   1:  PR[GP1:91,1] = PR[GP1:90,1] + 33.449;
   1:  PR[GP1:91,2] = PR[GP1:90,2] + -36.632;
   1:L PR[91] 10mm/sec CNT100;
   1:  PR[GP1:91,1] = PR[GP1:90,1] + 41.672;
   1:  PR[GP1:91,2] = PR[GP1:90,2] + -33.015;
   1:L PR[91] 10mm/sec CNT100;
   1:  PR[GP1:91,1] = PR[GP1:90,1] + 44.293;
   1:  PR[GP1:91,2] = PR[GP1:90,2] + -31.371;
   1:L PR[91] 10mm/sec CNT100;
   1:  PR[GP1:91,1] = PR[GP1:90,1] + 46.699;
   1:  PR[GP1:91,2] = PR[GP1:90,2] + -29.026;
   1:L PR[91] 10mm/sec CNT100;
   1:  PR[GP1:91,1] = PR[GP1:90,1] + 52.748;
   1:  PR[GP1:91,2] = PR[GP1:90,2] + -23.523;
   1:L PR[91] 10mm/sec CNT100;
   1:  PR[GP1:91,1] = PR[GP1:90,1] + 54.691;
   1:  PR[GP1:91,2] = PR[GP1:90,2] + -20.511;
   1:L PR[91] 10mm/sec CNT100;
   1:  PR[GP1:91,1] = PR[GP1:90,1] + 58.358;
   1:  PR[GP1:91,2] = PR[GP1:90,2] + -13.882;
   1:L PR[91] 10mm/sec CNT100;
   1:  PR[GP1:91,1] = PR[GP1:90,1] + 59.590;
   1:  PR[GP1:91,2] = PR[GP1:90,2] + -10.532;
   1:L PR[91] 10mm/sec CNT100;
   1:  PR[GP1:91,1] = PR[GP1:90,1] + 60.008;
   1:  PR[GP1:91,2] = PR[GP1:90,2] + -6.857;
   1:L PR[91] 10mm/sec CNT100;
   1:  PR[GP1:91,1] = PR[GP1:90,1] + 61.228;
   1:  PR[GP1:91,2] = PR[GP1:90,2] + 0.296;
   1:L PR[91] 10mm/sec CNT100;
   1:  PR[GP1:91,1] = PR[GP1:90,1] + 60.818;
   1:  PR[GP1:91,2] = PR[GP1:90,2] + 3.922;
   1:L PR[91] 10mm/sec CNT100;
   1:  PR[GP1:91,1] = PR[GP1:90,1] + 59.591;
   1:  PR[GP1:91,2] = PR[GP1:90,2] + 11.088;
   1:L PR[91] 10mm/sec CNT100;
   1:  PR[GP1:91,1] = PR[GP1:90,1] + 58.352;
   1:  PR[GP1:91,2] = PR[GP1:90,2] + 14.455;
   1:L PR[91] 10mm/sec CNT100;
   1:  PR[GP1:91,1] = PR[GP1:90,1] + 54.670;
   1:  PR[GP1:91,2] = PR[GP1:90,2] + 21.095;
   1:L PR[91] 10mm/sec CNT100;
   1:  PR[GP1:91,1] = PR[GP1:90,1] + 52.721;
   1:  PR[GP1:91,2] = PR[GP1:90,2] + 24.118;
   1:L PR[91] 10mm/sec CNT100;
   1:  PR[GP1:91,1] = PR[GP1:90,1] + 50.377;
   1:  PR[GP1:91,2] = PR[GP1:90,2] + 26.413;
   1:L PR[91] 10mm/sec CNT100;
   1:  PR[GP1:91,1] = PR[GP1:90,1] + 44.256;
   1:  PR[GP1:91,2] = PR[GP1:90,2] + 31.953;
   1:L PR[91] 10mm/sec CNT100;
   1:  PR[GP1:91,1] = PR[GP1:90,1] + 41.625;
   1:  PR[GP1:91,2] = PR[GP1:90,2] + 33.604;
   1:L PR[91] 10mm/sec CNT100;
   1:  PR[GP1:91,1] = PR[GP1:90,1] + 33.371;
   1:  PR[GP1:91,2] = PR[GP1:90,2] + 37.210;
   1:L PR[91] 10mm/sec CNT100;
   1:  PR[GP1:91,1] = PR[GP1:90,1] + 30.668;
   1:  PR[GP1:91,2] = PR[GP1:90,2] + 38.196;
   1:L PR[91] 10mm/sec CNT100;
   1:  PR[GP1:91,1] = PR[GP1:90,1] + 28.112;
   1:  PR[GP1:91,2] = PR[GP1:90,2] + 38.559;
   1:L PR[91] 10mm/sec CNT100;
   1:  PR[GP1:91,1] = PR[GP1:90,1] + 18.357;
   1:  PR[GP1:91,2] = PR[GP1:90,2] + 39.465;
   1:L PR[91] 10mm/sec CNT100;
   1:  PR[GP1:91,1] = PR[GP1:90,1] + 16.104;
   1:  PR[GP1:91,2] = PR[GP1:90,2] + 39.316;
   1:L PR[91] 10mm/sec CNT100;
   1:  PR[GP1:91,1] = PR[GP1:90,1] + 5.716;
   1:  PR[GP1:91,2] = PR[GP1:90,2] + 36.862;
   1:L PR[91] 10mm/sec CNT100;
   1:  PR[GP1:91,1] = PR[GP1:90,1] + 3.913;
   1:  PR[GP1:91,2] = PR[GP1:90,2] + 36.344;
   1:L PR[91] 10mm/sec CNT100;
   1:  PR[GP1:91,1] = PR[GP1:90,1] + 1.574;
   1:  PR[GP1:91,2] = PR[GP1:90,2] + 35.102;
   1:L PR[91] 10mm/sec CNT100;
   1:  PR[GP1:91,1] = PR[GP1:90,1] + -0.263;
   1:  PR[GP1:91,2] = PR[GP1:90,2] + 33.609;
   1:L PR[91] 10mm/sec CNT100;
   1:  PR[GP1:91,1] = PR[GP1:90,1] + -2.096;
   1:  PR[GP1:91,2] = PR[GP1:90,2] + 35.099;
   1:L PR[91] 10mm/sec CNT100;
   1:  PR[GP1:91,1] = PR[GP1:90,1] + -4.438;
   1:  PR[GP1:91,2] = PR[GP1:90,2] + 36.345;
   1:L PR[91] 10mm/sec CNT100;
   1:  PR[GP1:91,1] = PR[GP1:90,1] + -6.237;
   1:  PR[GP1:91,2] = PR[GP1:90,2] + 36.862;
   1:L PR[91] 10mm/sec CNT100;
   1:  PR[GP1:91,1] = PR[GP1:90,1] + -16.629;
   1:  PR[GP1:91,2] = PR[GP1:90,2] + 39.315;
   1:L PR[91] 10mm/sec CNT100;
   1:  PR[GP1:91,1] = PR[GP1:90,1] + -18.875;
   1:  PR[GP1:91,2] = PR[GP1:90,2] + 39.464;
   1:L PR[91] 10mm/sec CNT100;
   1:  PR[GP1:91,1] = PR[GP1:90,1] + -21.435;
   1:  PR[GP1:91,2] = PR[GP1:90,2] + 39.109;
   1:L PR[91] 10mm/sec CNT100;
   1:  PR[GP1:91,1] = PR[GP1:90,1] + -31.222;
   1:  PR[GP1:91,2] = PR[GP1:90,2] + 38.189;
   1:L PR[91] 10mm/sec CNT100;
   1:  PR[GP1:91,1] = PR[GP1:90,1] + -33.908;
   1:  PR[GP1:91,2] = PR[GP1:90,2] + 37.206;
   1:L PR[91] 10mm/sec CNT100;
   1:  PR[GP1:91,1] = PR[GP1:90,1] + -42.162;
   1:  PR[GP1:91,2] = PR[GP1:90,2] + 33.597;
   1:L PR[91] 10mm/sec CNT100;
   1:  PR[GP1:91,1] = PR[GP1:90,1] + -44.799;
   1:  PR[GP1:91,2] = PR[GP1:90,2] + 31.934;
   1:L PR[91] 10mm/sec CNT100;
   1:  PR[GP1:91,1] = PR[GP1:90,1] + -47.210;
   1:  PR[GP1:91,2] = PR[GP1:90,2] + 29.580;
   1:L PR[91] 10mm/sec CNT100;
   1:  PR[GP1:91,1] = PR[GP1:90,1] + -53.284;
   1:  PR[GP1:91,2] = PR[GP1:90,2] + 24.081;
   1:L PR[91] 10mm/sec CNT100;
   1:  PR[GP1:91,1] = PR[GP1:90,1] + -55.205;
   1:  PR[GP1:91,2] = PR[GP1:90,2] + 21.082;
   1:L PR[91] 10mm/sec CNT100;
   1:  PR[GP1:91,1] = PR[GP1:90,1] + -58.888;
   1:  PR[GP1:91,2] = PR[GP1:90,2] + 14.430;
   1:L PR[91] 10mm/sec CNT100;
   1:  PR[GP1:91,1] = PR[GP1:90,1] + -60.126;
   1:  PR[GP1:91,2] = PR[GP1:90,2] + 11.020;
   1:L PR[91] 10mm/sec CNT100;
   1:  PR[GP1:91,1] = PR[GP1:90,1] + -60.529;
   1:  PR[GP1:91,2] = PR[GP1:90,2] + 7.423;
   1:L PR[91] 10mm/sec CNT100;
   1:  PR[GP1:91,1] = PR[GP1:90,1] + -61.754;
   1:  PR[GP1:91,2] = PR[GP1:90,2] + 0.261;
   1:L PR[91] 10mm/sec CNT100;
   1:  PR[GP1:91,1] = PR[GP1:90,1] + -61.359;
   1:  PR[GP1:91,2] = PR[GP1:90,2] + -3.287;
   1:L PR[91] 10mm/sec CNT100;
   1:  PR[GP1:91,1] = PR[GP1:90,1] + -60.137;
   1:  PR[GP1:91,2] = PR[GP1:90,2] + -10.430;
   1:L PR[91] 10mm/sec CNT100;
   1:  PR[GP1:91,1] = PR[GP1:90,1] + -58.893;
   1:  PR[GP1:91,2] = PR[GP1:90,2] + -13.857;
   1:L PR[91] 10mm/sec CNT100;
   1:  PR[GP1:91,1] = PR[GP1:90,1] + -55.226;
   1:  PR[GP1:91,2] = PR[GP1:90,2] + -20.497;
   1:L PR[91] 10mm/sec CNT100;
   1:  PR[GP1:91,1] = PR[GP1:90,1] + -53.299;
   1:  PR[GP1:91,2] = PR[GP1:90,2] + -23.506;
   1:L PR[91] 10mm/sec CNT100;
   1:  PR[GP1:91,1] = PR[GP1:90,1] + -50.951;
   1:  PR[GP1:91,2] = PR[GP1:90,2] + -25.809;
   1:L PR[91] 10mm/sec CNT100;
   1:  PR[GP1:91,1] = PR[GP1:90,1] + -44.856;
   1:  PR[GP1:91,2] = PR[GP1:90,2] + -31.339;
   1:L PR[91] 10mm/sec CNT100;
   1:  PR[GP1:91,1] = PR[GP1:90,1] + -42.208;
   1:  PR[GP1:91,2] = PR[GP1:90,2] + -33.008;
   1:L PR[91] 10mm/sec CNT100;
   1:  PR[GP1:91,1] = PR[GP1:90,1] + -33.986;
   1:  PR[GP1:91,2] = PR[GP1:90,2] + -36.627;
   1:L PR[91] 10mm/sec CNT100;
   1:  PR[GP1:91,1] = PR[GP1:90,1] + -31.287;
   1:  PR[GP1:91,2] = PR[GP1:90,2] + -37.616;
   1:L PR[91] 10mm/sec CNT100;
   1:  PR[GP1:91,1] = PR[GP1:90,1] + -28.722;
   1:  PR[GP1:91,2] = PR[GP1:90,2] + -37.981;
   1:L PR[91] 10mm/sec CNT100;
   1:  PR[GP1:91,1] = PR[GP1:90,1] + -18.999;
   1:  PR[GP1:91,2] = PR[GP1:90,2] + -38.913;
   1:L PR[91] 10mm/sec CNT100;
   1:  PR[GP1:91,1] = PR[GP1:90,1] + -16.737;
   1:  PR[GP1:91,2] = PR[GP1:90,2] + -38.764;
   1:L PR[91] 10mm/sec CNT100;
   1:  PR[GP1:91,1] = PR[GP1:90,1] + -6.516;
   1:  PR[GP1:91,2] = PR[GP1:90,2] + -36.426;
   1:L PR[91] 10mm/sec CNT100;
   1:  PR[GP1:91,1] = PR[GP1:90,1] + -4.644;
   1:  PR[GP1:91,2] = PR[GP1:90,2] + -35.888;
   1:L PR[91] 10mm/sec CNT100;
   1:  PR[GP1:91,1] = PR[GP1:90,1] + -0.265;
   1:  PR[GP1:91,2] = PR[GP1:90,2] + -33.323;
   1:L PR[91] 10mm/sec CNT100;
   1:  PR[GP1:91,1] = PR[GP1:90,1] + 3.860;
   1:  PR[GP1:91,2] = PR[GP1:90,2] + -35.957;
   1:  PR[GP1:91,3] = PR[GP1:90,3] + 75.335;
   1:L PR[91] 10mm/sec CNT100;
   1:  PR[GP1:91,1] = PR[GP1:90,1] + 5.615;
   1:  PR[GP1:91,2] = PR[GP1:90,2] + -36.460;
   1:L PR[91] 10mm/sec CNT100;
   1:  PR[GP1:91,1] = PR[GP1:90,1] + 16.035;
   1:  PR[GP1:91,2] = PR[GP1:90,2] + -38.845;
   1:L PR[91] 10mm/sec CNT100;
   1:  PR[GP1:91,1] = PR[GP1:90,1] + 18.154;
   1:  PR[GP1:91,2] = PR[GP1:90,2] + -38.985;
   1:L PR[91] 10mm/sec CNT100;
   1:  PR[GP1:91,1] = PR[GP1:90,1] + 20.568;
   1:  PR[GP1:91,2] = PR[GP1:90,2] + -38.652;
   1:L PR[91] 10mm/sec CNT100;
   1:  PR[GP1:91,1] = PR[GP1:90,1] + 30.542;
   1:  PR[GP1:91,2] = PR[GP1:90,2] + -37.683;
   1:L PR[91] 10mm/sec CNT100;
   1:  PR[GP1:91,1] = PR[GP1:90,1] + 33.105;
   1:  PR[GP1:91,2] = PR[GP1:90,2] + -36.747;
   1:L PR[91] 10mm/sec CNT100;
   1:  PR[GP1:91,1] = PR[GP1:90,1] + 41.526;
   1:  PR[GP1:91,2] = PR[GP1:90,2] + -33.044;
   1:L PR[91] 10mm/sec CNT100;
   1:  PR[GP1:91,1] = PR[GP1:90,1] + 44.038;
   1:  PR[GP1:91,2] = PR[GP1:90,2] + -31.468;
   1:L PR[91] 10mm/sec CNT100;
   1:  PR[GP1:91,1] = PR[GP1:90,1] + 46.343;
   1:  PR[GP1:91,2] = PR[GP1:90,2] + -29.221;
   1:L PR[91] 10mm/sec CNT100;
   1:  PR[GP1:91,1] = PR[GP1:90,1] + 52.561;
   1:  PR[GP1:91,2] = PR[GP1:90,2] + -23.565;
   1:L PR[91] 10mm/sec CNT100;
   1:  PR[GP1:91,1] = PR[GP1:90,1] + 54.429;
   1:  PR[GP1:91,2] = PR[GP1:90,2] + -20.668;
   1:L PR[91] 10mm/sec CNT100;
   1:  PR[GP1:91,1] = PR[GP1:90,1] + 58.203;
   1:  PR[GP1:91,2] = PR[GP1:90,2] + -13.846;
   1:L PR[91] 10mm/sec CNT100;
   1:  PR[GP1:91,1] = PR[GP1:90,1] + 59.390;
   1:  PR[GP1:91,2] = PR[GP1:90,2] + -10.618;
   1:L PR[91] 10mm/sec CNT100;
   1:  PR[GP1:91,1] = PR[GP1:90,1] + 59.793;
   1:  PR[GP1:91,2] = PR[GP1:90,2] + -7.077;
   1:L PR[91] 10mm/sec CNT100;
   1:  PR[GP1:91,1] = PR[GP1:90,1] + 61.050;
   1:  PR[GP1:91,2] = PR[GP1:90,2] + 0.296;
   1:L PR[91] 10mm/sec CNT100;
   1:  PR[GP1:91,1] = PR[GP1:90,1] + 60.655;
   1:  PR[GP1:91,2] = PR[GP1:90,2] + 3.792;
   1:L PR[91] 10mm/sec CNT100;
   1:  PR[GP1:91,1] = PR[GP1:90,1] + 59.391;
   1:  PR[GP1:91,2] = PR[GP1:90,2] + 11.176;
   1:L PR[91] 10mm/sec CNT100;
   1:  PR[GP1:91,1] = PR[GP1:90,1] + 58.198;
   1:  PR[GP1:91,2] = PR[GP1:90,2] + 14.419;
   1:L PR[91] 10mm/sec CNT100;
   1:  PR[GP1:91,1] = PR[GP1:90,1] + 54.407;
   1:  PR[GP1:91,2] = PR[GP1:90,2] + 21.254;
   1:L PR[91] 10mm/sec CNT100;
   1:  PR[GP1:91,1] = PR[GP1:90,1] + 52.534;
   1:  PR[GP1:91,2] = PR[GP1:90,2] + 24.160;
   1:L PR[91] 10mm/sec CNT100;
   1:  PR[GP1:91,1] = PR[GP1:90,1] + 50.279;
   1:  PR[GP1:91,2] = PR[GP1:90,2] + 26.367;
   1:L PR[91] 10mm/sec CNT100;
   1:  PR[GP1:91,1] = PR[GP1:90,1] + 43.999;
   1:  PR[GP1:91,2] = PR[GP1:90,2] + 32.051;
   1:L PR[91] 10mm/sec CNT100;
   1:  PR[GP1:91,1] = PR[GP1:90,1] + 41.479;
   1:  PR[GP1:91,2] = PR[GP1:90,2] + 33.633;
   1:L PR[91] 10mm/sec CNT100;
   1:  PR[GP1:91,1] = PR[GP1:90,1] + 33.025;
   1:  PR[GP1:91,2] = PR[GP1:90,2] + 37.326;
   1:L PR[91] 10mm/sec CNT100;
   1:  PR[GP1:91,1] = PR[GP1:90,1] + 30.449;
   1:  PR[GP1:91,2] = PR[GP1:90,2] + 38.266;
   1:L PR[91] 10mm/sec CNT100;
   1:  PR[GP1:91,1] = PR[GP1:90,1] + 28.013;
   1:  PR[GP1:91,2] = PR[GP1:90,2] + 38.612;
   1:L PR[91] 10mm/sec CNT100;
   1:  PR[GP1:91,1] = PR[GP1:90,1] + 18.055;
   1:  PR[GP1:91,2] = PR[GP1:90,2] + 39.537;
   1:L PR[91] 10mm/sec CNT100;
   1:  PR[GP1:91,1] = PR[GP1:90,1] + 15.925;
   1:  PR[GP1:91,2] = PR[GP1:90,2] + 39.396;
   1:L PR[91] 10mm/sec CNT100;
   1:  PR[GP1:91,1] = PR[GP1:90,1] + 5.335;
   1:  PR[GP1:91,2] = PR[GP1:90,2] + 36.894;
   1:L PR[91] 10mm/sec CNT100;
   1:  PR[GP1:91,1] = PR[GP1:90,1] + 3.655;
   1:  PR[GP1:91,2] = PR[GP1:90,2] + 36.412;
   1:L PR[91] 10mm/sec CNT100;
   1:  PR[GP1:91,1] = PR[GP1:90,1] + 1.401;
   1:  PR[GP1:91,2] = PR[GP1:90,2] + 35.217;
   1:L PR[91] 10mm/sec CNT100;
   1:  PR[GP1:91,1] = PR[GP1:90,1] + -0.263;
   1:  PR[GP1:91,2] = PR[GP1:90,2] + 33.863;
   1:L PR[91] 10mm/sec CNT100;
   1:  PR[GP1:91,1] = PR[GP1:90,1] + -1.924;
   1:  PR[GP1:91,2] = PR[GP1:90,2] + 35.213;
   1:L PR[91] 10mm/sec CNT100;
   1:  PR[GP1:91,1] = PR[GP1:90,1] + -4.180;
   1:  PR[GP1:91,2] = PR[GP1:90,2] + 36.412;
   1:L PR[91] 10mm/sec CNT100;
   1:  PR[GP1:91,1] = PR[GP1:90,1] + -5.857;
   1:  PR[GP1:91,2] = PR[GP1:90,2] + 36.895;
   1:L PR[91] 10mm/sec CNT100;
   1:  PR[GP1:91,1] = PR[GP1:90,1] + -16.450;
   1:  PR[GP1:91,2] = PR[GP1:90,2] + 39.395;
   1:L PR[91] 10mm/sec CNT100;
   1:  PR[GP1:91,1] = PR[GP1:90,1] + -18.573;
   1:  PR[GP1:91,2] = PR[GP1:90,2] + 39.536;
   1:L PR[91] 10mm/sec CNT100;
   1:  PR[GP1:91,1] = PR[GP1:90,1] + -20.996;
   1:  PR[GP1:91,2] = PR[GP1:90,2] + 39.200;
   1:L PR[91] 10mm/sec CNT100;
   1:  PR[GP1:91,1] = PR[GP1:90,1] + -31.002;
   1:  PR[GP1:91,2] = PR[GP1:90,2] + 38.260;
   1:L PR[91] 10mm/sec CNT100;
   1:  PR[GP1:91,1] = PR[GP1:90,1] + -33.561;
   1:  PR[GP1:91,2] = PR[GP1:90,2] + 37.322;
   1:L PR[91] 10mm/sec CNT100;
   1:  PR[GP1:91,1] = PR[GP1:90,1] + -42.015;
   1:  PR[GP1:91,2] = PR[GP1:90,2] + 33.626;
   1:L PR[91] 10mm/sec CNT100;
   1:  PR[GP1:91,1] = PR[GP1:90,1] + -44.541;
   1:  PR[GP1:91,2] = PR[GP1:90,2] + 32.033;
   1:L PR[91] 10mm/sec CNT100;
   1:  PR[GP1:91,1] = PR[GP1:90,1] + -46.852;
   1:  PR[GP1:91,2] = PR[GP1:90,2] + 29.777;
   1:L PR[91] 10mm/sec CNT100;
   1:  PR[GP1:91,1] = PR[GP1:90,1] + -53.096;
   1:  PR[GP1:91,2] = PR[GP1:90,2] + 24.124;
   1:L PR[91] 10mm/sec CNT100;
   1:  PR[GP1:91,1] = PR[GP1:90,1] + -54.943;
   1:  PR[GP1:91,2] = PR[GP1:90,2] + 21.241;
   1:L PR[91] 10mm/sec CNT100;
   1:  PR[GP1:91,1] = PR[GP1:90,1] + -58.733;
   1:  PR[GP1:91,2] = PR[GP1:90,2] + 14.394;
   1:L PR[91] 10mm/sec CNT100;
   1:  PR[GP1:91,1] = PR[GP1:90,1] + -59.925;
   1:  PR[GP1:91,2] = PR[GP1:90,2] + 11.110;
   1:L PR[91] 10mm/sec CNT100;
   1:  PR[GP1:91,1] = PR[GP1:90,1] + -60.314;
   1:  PR[GP1:91,2] = PR[GP1:90,2] + 7.643;
   1:L PR[91] 10mm/sec CNT100;
   1:  PR[GP1:91,1] = PR[GP1:90,1] + -61.577;
   1:  PR[GP1:91,2] = PR[GP1:90,2] + 0.261;
   1:L PR[91] 10mm/sec CNT100;
   1:  PR[GP1:91,1] = PR[GP1:90,1] + -61.196;
   1:  PR[GP1:91,2] = PR[GP1:90,2] + -3.159;
   1:L PR[91] 10mm/sec CNT100;
   1:  PR[GP1:91,1] = PR[GP1:90,1] + -59.937;
   1:  PR[GP1:91,2] = PR[GP1:90,2] + -10.520;
   1:L PR[91] 10mm/sec CNT100;
   1:  PR[GP1:91,1] = PR[GP1:90,1] + -58.739;
   1:  PR[GP1:91,2] = PR[GP1:90,2] + -13.821;
   1:L PR[91] 10mm/sec CNT100;
   1:  PR[GP1:91,1] = PR[GP1:90,1] + -54.964;
   1:  PR[GP1:91,2] = PR[GP1:90,2] + -20.656;
   1:L PR[91] 10mm/sec CNT100;
   1:  PR[GP1:91,1] = PR[GP1:90,1] + -53.111;
   1:  PR[GP1:91,2] = PR[GP1:90,2] + -23.549;
   1:L PR[91] 10mm/sec CNT100;
   1:  PR[GP1:91,1] = PR[GP1:90,1] + -50.853;
   1:  PR[GP1:91,2] = PR[GP1:90,2] + -25.764;
   1:L PR[91] 10mm/sec CNT100;
   1:  PR[GP1:91,1] = PR[GP1:90,1] + -44.599;
   1:  PR[GP1:91,2] = PR[GP1:90,2] + -31.438;
   1:L PR[91] 10mm/sec CNT100;
   1:  PR[GP1:91,1] = PR[GP1:90,1] + -42.063;
   1:  PR[GP1:91,2] = PR[GP1:90,2] + -33.037;
   1:L PR[91] 10mm/sec CNT100;
   1:  PR[GP1:91,1] = PR[GP1:90,1] + -33.642;
   1:  PR[GP1:91,2] = PR[GP1:90,2] + -36.743;
   1:L PR[91] 10mm/sec CNT100;
   1:  PR[GP1:91,1] = PR[GP1:90,1] + -31.069;
   1:  PR[GP1:91,2] = PR[GP1:90,2] + -37.685;
   1:L PR[91] 10mm/sec CNT100;
   1:  PR[GP1:91,1] = PR[GP1:90,1] + -28.624;
   1:  PR[GP1:91,2] = PR[GP1:90,2] + -38.033;
   1:L PR[91] 10mm/sec CNT100;
   1:  PR[GP1:91,1] = PR[GP1:90,1] + -18.699;
   1:  PR[GP1:91,2] = PR[GP1:90,2] + -38.985;
   1:L PR[91] 10mm/sec CNT100;
   1:  PR[GP1:91,1] = PR[GP1:90,1] + -16.560;
   1:  PR[GP1:91,2] = PR[GP1:90,2] + -38.844;
   1:L PR[91] 10mm/sec CNT100;
   1:  PR[GP1:91,1] = PR[GP1:90,1] + -6.141;
   1:  PR[GP1:91,2] = PR[GP1:90,2] + -36.461;
   1:L PR[91] 10mm/sec CNT100;
   1:  PR[GP1:91,1] = PR[GP1:90,1] + -4.389;
   1:  PR[GP1:91,2] = PR[GP1:90,2] + -35.957;
   1:L PR[91] 10mm/sec CNT100;
   1:  PR[GP1:91,1] = PR[GP1:90,1] + -0.265;
   1:  PR[GP1:91,2] = PR[GP1:90,2] + -33.542;
   1:L PR[91] 10mm/sec CNT100;
   1:  PR[GP1:91,1] = PR[GP1:90,1] + 3.606;
   1:  PR[GP1:91,2] = PR[GP1:90,2] + -36.026;
   1:  PR[GP1:91,3] = PR[GP1:90,3] + 75.945;
   1:L PR[91] 10mm/sec CNT100;
   1:  PR[GP1:91,1] = PR[GP1:90,1] + 5.240;
   1:  PR[GP1:91,2] = PR[GP1:90,2] + -36.495;
   1:L PR[91] 10mm/sec CNT100;
   1:  PR[GP1:91,1] = PR[GP1:90,1] + 15.858;
   1:  PR[GP1:91,2] = PR[GP1:90,2] + -38.925;
   1:L PR[91] 10mm/sec CNT100;
   1:  PR[GP1:91,1] = PR[GP1:90,1] + 17.854;
   1:  PR[GP1:91,2] = PR[GP1:90,2] + -39.057;
   1:L PR[91] 10mm/sec CNT100;
   1:  PR[GP1:91,1] = PR[GP1:90,1] + 20.132;
   1:  PR[GP1:91,2] = PR[GP1:90,2] + -38.743;
   1:L PR[91] 10mm/sec CNT100;
   1:  PR[GP1:91,1] = PR[GP1:90,1] + 30.324;
   1:  PR[GP1:91,2] = PR[GP1:90,2] + -37.752;
   1:L PR[91] 10mm/sec CNT100;
   1:  PR[GP1:91,1] = PR[GP1:90,1] + 32.761;
   1:  PR[GP1:91,2] = PR[GP1:90,2] + -36.863;
   1:L PR[91] 10mm/sec CNT100;
   1:  PR[GP1:91,1] = PR[GP1:90,1] + 41.381;
   1:  PR[GP1:91,2] = PR[GP1:90,2] + -33.072;
   1:L PR[91] 10mm/sec CNT100;
   1:  PR[GP1:91,1] = PR[GP1:90,1] + 43.782;
   1:  PR[GP1:91,2] = PR[GP1:90,2] + -31.566;
   1:L PR[91] 10mm/sec CNT100;
   1:  PR[GP1:91,1] = PR[GP1:90,1] + 45.988;
   1:  PR[GP1:91,2] = PR[GP1:90,2] + -29.415;
   1:L PR[91] 10mm/sec CNT100;
   1:  PR[GP1:91,1] = PR[GP1:90,1] + 52.375;
   1:  PR[GP1:91,2] = PR[GP1:90,2] + -23.606;
   1:L PR[91] 10mm/sec CNT100;
   1:  PR[GP1:91,1] = PR[GP1:90,1] + 54.167;
   1:  PR[GP1:91,2] = PR[GP1:90,2] + -20.826;
   1:L PR[91] 10mm/sec CNT100;
   1:  PR[GP1:91,1] = PR[GP1:90,1] + 58.049;
   1:  PR[GP1:91,2] = PR[GP1:90,2] + -13.809;
   1:L PR[91] 10mm/sec CNT100;
   1:  PR[GP1:91,1] = PR[GP1:90,1] + 59.191;
   1:  PR[GP1:91,2] = PR[GP1:90,2] + -10.705;
   1:L PR[91] 10mm/sec CNT100;
   1:  PR[GP1:91,1] = PR[GP1:90,1] + 59.578;
   1:  PR[GP1:91,2] = PR[GP1:90,2] + -7.297;
   1:L PR[91] 10mm/sec CNT100;
   1:  PR[GP1:91,1] = PR[GP1:90,1] + 60.873;
   1:  PR[GP1:91,2] = PR[GP1:90,2] + 0.296;
   1:L PR[91] 10mm/sec CNT100;
   1:  PR[GP1:91,1] = PR[GP1:90,1] + 60.493;
   1:  PR[GP1:91,2] = PR[GP1:90,2] + 3.661;
   1:L PR[91] 10mm/sec CNT100;
   1:  PR[GP1:91,1] = PR[GP1:90,1] + 59.191;
   1:  PR[GP1:91,2] = PR[GP1:90,2] + 11.263;
   1:L PR[91] 10mm/sec CNT100;
   1:  PR[GP1:91,1] = PR[GP1:90,1] + 58.044;
   1:  PR[GP1:91,2] = PR[GP1:90,2] + 14.382;
   1:L PR[91] 10mm/sec CNT100;
   1:  PR[GP1:91,1] = PR[GP1:90,1] + 54.145;
   1:  PR[GP1:91,2] = PR[GP1:90,2] + 21.412;
   1:L PR[91] 10mm/sec CNT100;
   1:  PR[GP1:91,1] = PR[GP1:90,1] + 52.346;
   1:  PR[GP1:91,2] = PR[GP1:90,2] + 24.202;
   1:L PR[91] 10mm/sec CNT100;
   1:  PR[GP1:91,1] = PR[GP1:90,1] + 50.182;
   1:  PR[GP1:91,2] = PR[GP1:90,2] + 26.322;
   1:L PR[91] 10mm/sec CNT100;
   1:  PR[GP1:91,1] = PR[GP1:90,1] + 43.742;
   1:  PR[GP1:91,2] = PR[GP1:90,2] + 32.150;
   1:L PR[91] 10mm/sec CNT100;
   1:  PR[GP1:91,1] = PR[GP1:90,1] + 41.332;
   1:  PR[GP1:91,2] = PR[GP1:90,2] + 33.662;
   1:L PR[91] 10mm/sec CNT100;
   1:  PR[GP1:91,1] = PR[GP1:90,1] + 32.679;
   1:  PR[GP1:91,2] = PR[GP1:90,2] + 37.443;
   1:L PR[91] 10mm/sec CNT100;
   1:  PR[GP1:91,1] = PR[GP1:90,1] + 30.230;
   1:  PR[GP1:91,2] = PR[GP1:90,2] + 38.336;
   1:L PR[91] 10mm/sec CNT100;
   1:  PR[GP1:91,1] = PR[GP1:90,1] + 27.913;
   1:  PR[GP1:91,2] = PR[GP1:90,2] + 38.665;
   1:L PR[91] 10mm/sec CNT100;
   1:  PR[GP1:91,1] = PR[GP1:90,1] + 17.753;
   1:  PR[GP1:91,2] = PR[GP1:90,2] + 39.609;
   1:L PR[91] 10mm/sec CNT100;
   1:  PR[GP1:91,1] = PR[GP1:90,1] + 15.746;
   1:  PR[GP1:91,2] = PR[GP1:90,2] + 39.476;
   1:L PR[91] 10mm/sec CNT100;
   1:  PR[GP1:91,1] = PR[GP1:90,1] + 4.954;
   1:  PR[GP1:91,2] = PR[GP1:90,2] + 36.927;
   1:L PR[91] 10mm/sec CNT100;
   1:  PR[GP1:91,1] = PR[GP1:90,1] + 3.397;
   1:  PR[GP1:91,2] = PR[GP1:90,2] + 36.479;
   1:L PR[91] 10mm/sec CNT100;
   1:  PR[GP1:91,1] = PR[GP1:90,1] + 1.228;
   1:  PR[GP1:91,2] = PR[GP1:90,2] + 35.330;
   1:L PR[91] 10mm/sec CNT100;
   1:  PR[GP1:91,1] = PR[GP1:90,1] + -0.263;
   1:  PR[GP1:91,2] = PR[GP1:90,2] + 34.118;
   1:L PR[91] 10mm/sec CNT100;
   1:  PR[GP1:91,1] = PR[GP1:90,1] + -1.751;
   1:  PR[GP1:91,2] = PR[GP1:90,2] + 35.328;
   1:L PR[91] 10mm/sec CNT100;
   1:  PR[GP1:91,1] = PR[GP1:90,1] + -3.921;
   1:  PR[GP1:91,2] = PR[GP1:90,2] + 36.480;
   1:L PR[91] 10mm/sec CNT100;
   1:  PR[GP1:91,1] = PR[GP1:90,1] + -5.476;
   1:  PR[GP1:91,2] = PR[GP1:90,2] + 36.927;
   1:L PR[91] 10mm/sec CNT100;
   1:  PR[GP1:91,1] = PR[GP1:90,1] + -16.271;
   1:  PR[GP1:91,2] = PR[GP1:90,2] + 39.475;
   1:L PR[91] 10mm/sec CNT100;
   1:  PR[GP1:91,1] = PR[GP1:90,1] + -18.270;
   1:  PR[GP1:91,2] = PR[GP1:90,2] + 39.607;
   1:L PR[91] 10mm/sec CNT100;
   1:  PR[GP1:91,1] = PR[GP1:90,1] + -20.556;
   1:  PR[GP1:91,2] = PR[GP1:90,2] + 39.291;
   1:L PR[91] 10mm/sec CNT100;
   1:  PR[GP1:91,1] = PR[GP1:90,1] + -30.782;
   1:  PR[GP1:91,2] = PR[GP1:90,2] + 38.330;
   1:L PR[91] 10mm/sec CNT100;
   1:  PR[GP1:91,1] = PR[GP1:90,1] + -33.215;
   1:  PR[GP1:91,2] = PR[GP1:90,2] + 37.439;
   1:L PR[91] 10mm/sec CNT100;
   1:  PR[GP1:91,1] = PR[GP1:90,1] + -41.868;
   1:  PR[GP1:91,2] = PR[GP1:90,2] + 33.655;
   1:L PR[91] 10mm/sec CNT100;
   1:  PR[GP1:91,1] = PR[GP1:90,1] + -44.283;
   1:  PR[GP1:91,2] = PR[GP1:90,2] + 32.132;
   1:L PR[91] 10mm/sec CNT100;
   1:  PR[GP1:91,1] = PR[GP1:90,1] + -46.495;
   1:  PR[GP1:91,2] = PR[GP1:90,2] + 29.974;
   1:L PR[91] 10mm/sec CNT100;
   1:  PR[GP1:91,1] = PR[GP1:90,1] + -52.907;
   1:  PR[GP1:91,2] = PR[GP1:90,2] + 24.168;
   1:L PR[91] 10mm/sec CNT100;
   1:  PR[GP1:91,1] = PR[GP1:90,1] + -54.680;
   1:  PR[GP1:91,2] = PR[GP1:90,2] + 21.401;
   1:L PR[91] 10mm/sec CNT100;
   1:  PR[GP1:91,1] = PR[GP1:90,1] + -58.579;
   1:  PR[GP1:91,2] = PR[GP1:90,2] + 14.358;
   1:L PR[91] 10mm/sec CNT100;
   1:  PR[GP1:91,1] = PR[GP1:90,1] + -59.725;
   1:  PR[GP1:91,2] = PR[GP1:90,2] + 11.200;
   1:L PR[91] 10mm/sec CNT100;
   1:  PR[GP1:91,1] = PR[GP1:90,1] + -60.099;
   1:  PR[GP1:91,2] = PR[GP1:90,2] + 7.863;
   1:L PR[91] 10mm/sec CNT100;
   1:  PR[GP1:91,1] = PR[GP1:90,1] + -61.400;
   1:  PR[GP1:91,2] = PR[GP1:90,2] + 0.261;
   1:L PR[91] 10mm/sec CNT100;
   1:  PR[GP1:91,1] = PR[GP1:90,1] + -61.033;
   1:  PR[GP1:91,2] = PR[GP1:90,2] + -3.031;
   1:L PR[91] 10mm/sec CNT100;
   1:  PR[GP1:91,1] = PR[GP1:90,1] + -59.737;
   1:  PR[GP1:91,2] = PR[GP1:90,2] + -10.609;
   1:L PR[91] 10mm/sec CNT100;
   1:  PR[GP1:91,1] = PR[GP1:90,1] + -58.584;
   1:  PR[GP1:91,2] = PR[GP1:90,2] + -13.785;
   1:L PR[91] 10mm/sec CNT100;
   1:  PR[GP1:91,1] = PR[GP1:90,1] + -54.702;
   1:  PR[GP1:91,2] = PR[GP1:90,2] + -20.814;
   1:L PR[91] 10mm/sec CNT100;
   1:  PR[GP1:91,1] = PR[GP1:90,1] + -52.923;
   1:  PR[GP1:91,2] = PR[GP1:90,2] + -23.592;
   1:L PR[91] 10mm/sec CNT100;
   1:  PR[GP1:91,1] = PR[GP1:90,1] + -50.755;
   1:  PR[GP1:91,2] = PR[GP1:90,2] + -25.718;
   1:L PR[91] 10mm/sec CNT100;
   1:  PR[GP1:91,1] = PR[GP1:90,1] + -44.342;
   1:  PR[GP1:91,2] = PR[GP1:90,2] + -31.536;
   1:L PR[91] 10mm/sec CNT100;
   1:  PR[GP1:91,1] = PR[GP1:90,1] + -41.917;
   1:  PR[GP1:91,2] = PR[GP1:90,2] + -33.065;
   1:L PR[91] 10mm/sec CNT100;
   1:  PR[GP1:91,1] = PR[GP1:90,1] + -33.297;
   1:  PR[GP1:91,2] = PR[GP1:90,2] + -36.859;
   1:L PR[91] 10mm/sec CNT100;
   1:  PR[GP1:91,1] = PR[GP1:90,1] + -30.851;
   1:  PR[GP1:91,2] = PR[GP1:90,2] + -37.755;
   1:L PR[91] 10mm/sec CNT100;
   1:  PR[GP1:91,1] = PR[GP1:90,1] + -28.527;
   1:  PR[GP1:91,2] = PR[GP1:90,2] + -38.086;
   1:L PR[91] 10mm/sec CNT100;
   1:  PR[GP1:91,1] = PR[GP1:90,1] + -18.398;
   1:  PR[GP1:91,2] = PR[GP1:90,2] + -39.057;
   1:L PR[91] 10mm/sec CNT100;
   1:  PR[GP1:91,1] = PR[GP1:90,1] + -16.383;
   1:  PR[GP1:91,2] = PR[GP1:90,2] + -38.925;
   1:L PR[91] 10mm/sec CNT100;
   1:  PR[GP1:91,1] = PR[GP1:90,1] + -5.765;
   1:  PR[GP1:91,2] = PR[GP1:90,2] + -36.495;
   1:L PR[91] 10mm/sec CNT100;
   1:  PR[GP1:91,1] = PR[GP1:90,1] + -4.134;
   1:  PR[GP1:91,2] = PR[GP1:90,2] + -36.027;
   1:L PR[91] 10mm/sec CNT100;
   1:  PR[GP1:91,1] = PR[GP1:90,1] + -0.265;
   1:  PR[GP1:91,2] = PR[GP1:90,2] + -33.760;
   1:L PR[91] 10mm/sec CNT100;
   1:  PR[GP1:91,1] = PR[GP1:90,1] + 3.351;
   1:  PR[GP1:91,2] = PR[GP1:90,2] + -36.095;
   1:  PR[GP1:91,3] = PR[GP1:90,3] + 76.555;
   1:L PR[91] 10mm/sec CNT100;
   1:  PR[GP1:91,1] = PR[GP1:90,1] + 4.864;
   1:  PR[GP1:91,2] = PR[GP1:90,2] + -36.530;
   1:L PR[91] 10mm/sec CNT100;
   1:  PR[GP1:91,1] = PR[GP1:90,1] + 15.681;
   1:  PR[GP1:91,2] = PR[GP1:90,2] + -39.005;
   1:L PR[91] 10mm/sec CNT100;
   1:  PR[GP1:91,1] = PR[GP1:90,1] + 17.554;
   1:  PR[GP1:91,2] = PR[GP1:90,2] + -39.129;
   1:L PR[91] 10mm/sec CNT100;
   1:  PR[GP1:91,1] = PR[GP1:90,1] + 19.696;
   1:  PR[GP1:91,2] = PR[GP1:90,2] + -38.834;
   1:L PR[91] 10mm/sec CNT100;
   1:  PR[GP1:91,1] = PR[GP1:90,1] + 30.107;
   1:  PR[GP1:91,2] = PR[GP1:90,2] + -37.822;
   1:L PR[91] 10mm/sec CNT100;
   1:  PR[GP1:91,1] = PR[GP1:90,1] + 32.417;
   1:  PR[GP1:91,2] = PR[GP1:90,2] + -36.979;
   1:L PR[91] 10mm/sec CNT100;
   1:  PR[GP1:91,1] = PR[GP1:90,1] + 41.236;
   1:  PR[GP1:91,2] = PR[GP1:90,2] + -33.100;
   1:L PR[91] 10mm/sec CNT100;
   1:  PR[GP1:91,1] = PR[GP1:90,1] + 43.526;
   1:  PR[GP1:91,2] = PR[GP1:90,2] + -31.663;
   1:L PR[91] 10mm/sec CNT100;
   1:  PR[GP1:91,1] = PR[GP1:90,1] + 45.633;
   1:  PR[GP1:91,2] = PR[GP1:90,2] + -29.610;
   1:L PR[91] 10mm/sec CNT100;
   1:  PR[GP1:91,1] = PR[GP1:90,1] + 52.188;
   1:  PR[GP1:91,2] = PR[GP1:90,2] + -23.648;
   1:L PR[91] 10mm/sec CNT100;
   1:  PR[GP1:91,1] = PR[GP1:90,1] + 53.905;
   1:  PR[GP1:91,2] = PR[GP1:90,2] + -20.984;
   1:L PR[91] 10mm/sec CNT100;
   1:  PR[GP1:91,1] = PR[GP1:90,1] + 57.895;
   1:  PR[GP1:91,2] = PR[GP1:90,2] + -13.772;
   1:L PR[91] 10mm/sec CNT100;
   1:  PR[GP1:91,1] = PR[GP1:90,1] + 58.991;
   1:  PR[GP1:91,2] = PR[GP1:90,2] + -10.792;
   1:L PR[91] 10mm/sec CNT100;
   1:  PR[GP1:91,1] = PR[GP1:90,1] + 59.363;
   1:  PR[GP1:91,2] = PR[GP1:90,2] + -7.517;
   1:L PR[91] 10mm/sec CNT100;
   1:  PR[GP1:91,1] = PR[GP1:90,1] + 60.696;
   1:  PR[GP1:91,2] = PR[GP1:90,2] + 0.296;
   1:L PR[91] 10mm/sec CNT100;
   1:  PR[GP1:91,1] = PR[GP1:90,1] + 60.330;
   1:  PR[GP1:91,2] = PR[GP1:90,2] + 3.530;
   1:L PR[91] 10mm/sec CNT100;
   1:  PR[GP1:91,1] = PR[GP1:90,1] + 58.991;
   1:  PR[GP1:91,2] = PR[GP1:90,2] + 11.350;
   1:L PR[91] 10mm/sec CNT100;
   1:  PR[GP1:91,1] = PR[GP1:90,1] + 57.890;
   1:  PR[GP1:91,2] = PR[GP1:90,2] + 14.346;
   1:L PR[91] 10mm/sec CNT100;
   1:  PR[GP1:91,1] = PR[GP1:90,1] + 53.883;
   1:  PR[GP1:91,2] = PR[GP1:90,2] + 21.570;
   1:L PR[91] 10mm/sec CNT100;
   1:  PR[GP1:91,1] = PR[GP1:90,1] + 52.159;
   1:  PR[GP1:91,2] = PR[GP1:90,2] + 24.245;
   1:L PR[91] 10mm/sec CNT100;
   1:  PR[GP1:91,1] = PR[GP1:90,1] + 50.085;
   1:  PR[GP1:91,2] = PR[GP1:90,2] + 26.276;
   1:L PR[91] 10mm/sec CNT100;
   1:  PR[GP1:91,1] = PR[GP1:90,1] + 43.485;
   1:  PR[GP1:91,2] = PR[GP1:90,2] + 32.248;
   1:L PR[91] 10mm/sec CNT100;
   1:  PR[GP1:91,1] = PR[GP1:90,1] + 41.186;
   1:  PR[GP1:91,2] = PR[GP1:90,2] + 33.691;
   1:L PR[91] 10mm/sec CNT100;
   1:  PR[GP1:91,1] = PR[GP1:90,1] + 32.333;
   1:  PR[GP1:91,2] = PR[GP1:90,2] + 37.559;
   1:L PR[91] 10mm/sec CNT100;
   1:  PR[GP1:91,1] = PR[GP1:90,1] + 30.010;
   1:  PR[GP1:91,2] = PR[GP1:90,2] + 38.406;
   1:L PR[91] 10mm/sec CNT100;
   1:  PR[GP1:91,1] = PR[GP1:90,1] + 27.814;
   1:  PR[GP1:91,2] = PR[GP1:90,2] + 38.718;
   1:L PR[91] 10mm/sec CNT100;
   1:  PR[GP1:91,1] = PR[GP1:90,1] + 17.450;
   1:  PR[GP1:91,2] = PR[GP1:90,2] + 39.681;
   1:L PR[91] 10mm/sec CNT100;
   1:  PR[GP1:91,1] = PR[GP1:90,1] + 15.567;
   1:  PR[GP1:91,2] = PR[GP1:90,2] + 39.556;
   1:L PR[91] 10mm/sec CNT100;
   1:  PR[GP1:91,1] = PR[GP1:90,1] + 4.573;
   1:  PR[GP1:91,2] = PR[GP1:90,2] + 36.959;
   1:L PR[91] 10mm/sec CNT100;
   1:  PR[GP1:91,1] = PR[GP1:90,1] + 3.139;
   1:  PR[GP1:91,2] = PR[GP1:90,2] + 36.547;
   1:L PR[91] 10mm/sec CNT100;
   1:  PR[GP1:91,1] = PR[GP1:90,1] + 1.055;
   1:  PR[GP1:91,2] = PR[GP1:90,2] + 35.444;
   1:L PR[91] 10mm/sec CNT100;
   1:  PR[GP1:91,1] = PR[GP1:90,1] + -0.263;
   1:  PR[GP1:91,2] = PR[GP1:90,2] + 34.373;
   1:L PR[91] 10mm/sec CNT100;
   1:  PR[GP1:91,1] = PR[GP1:90,1] + -1.579;
   1:  PR[GP1:91,2] = PR[GP1:90,2] + 35.442;
   1:L PR[91] 10mm/sec CNT100;
   1:  PR[GP1:91,1] = PR[GP1:90,1] + -3.663;
   1:  PR[GP1:91,2] = PR[GP1:90,2] + 36.548;
   1:L PR[91] 10mm/sec CNT100;
   1:  PR[GP1:91,1] = PR[GP1:90,1] + -5.095;
   1:  PR[GP1:91,2] = PR[GP1:90,2] + 36.959;
   1:L PR[91] 10mm/sec CNT100;
   1:  PR[GP1:91,1] = PR[GP1:90,1] + -16.092;
   1:  PR[GP1:91,2] = PR[GP1:90,2] + 39.556;
   1:L PR[91] 10mm/sec CNT100;
   1:  PR[GP1:91,1] = PR[GP1:90,1] + -17.968;
   1:  PR[GP1:91,2] = PR[GP1:90,2] + 39.679;
   1:L PR[91] 10mm/sec CNT100;
   1:  PR[GP1:91,1] = PR[GP1:90,1] + -20.117;
   1:  PR[GP1:91,2] = PR[GP1:90,2] + 39.382;
   1:L PR[91] 10mm/sec CNT100;
   1:  PR[GP1:91,1] = PR[GP1:90,1] + -30.562;
   1:  PR[GP1:91,2] = PR[GP1:90,2] + 38.400;
   1:L PR[91] 10mm/sec CNT100;
   1:  PR[GP1:91,1] = PR[GP1:90,1] + -32.868;
   1:  PR[GP1:91,2] = PR[GP1:90,2] + 37.555;
   1:L PR[91] 10mm/sec CNT100;
   1:  PR[GP1:91,1] = PR[GP1:90,1] + -41.721;
   1:  PR[GP1:91,2] = PR[GP1:90,2] + 33.684;
   1:L PR[91] 10mm/sec CNT100;
   1:  PR[GP1:91,1] = PR[GP1:90,1] + -44.025;
   1:  PR[GP1:91,2] = PR[GP1:90,2] + 32.232;
   1:L PR[91] 10mm/sec CNT100;
   1:  PR[GP1:91,1] = PR[GP1:90,1] + -46.137;
   1:  PR[GP1:91,2] = PR[GP1:90,2] + 30.170;
   1:L PR[91] 10mm/sec CNT100;
   1:  PR[GP1:91,1] = PR[GP1:90,1] + -52.718;
   1:  PR[GP1:91,2] = PR[GP1:90,2] + 24.212;
   1:L PR[91] 10mm/sec CNT100;
   1:  PR[GP1:91,1] = PR[GP1:90,1] + -54.417;
   1:  PR[GP1:91,2] = PR[GP1:90,2] + 21.560;
   1:L PR[91] 10mm/sec CNT100;
   1:  PR[GP1:91,1] = PR[GP1:90,1] + -58.424;
   1:  PR[GP1:91,2] = PR[GP1:90,2] + 14.322;
   1:L PR[91] 10mm/sec CNT100;
   1:  PR[GP1:91,1] = PR[GP1:90,1] + -59.525;
   1:  PR[GP1:91,2] = PR[GP1:90,2] + 11.289;
   1:L PR[91] 10mm/sec CNT100;
   1:  PR[GP1:91,1] = PR[GP1:90,1] + -59.884;
   1:  PR[GP1:91,2] = PR[GP1:90,2] + 8.083;
   1:L PR[91] 10mm/sec CNT100;
   1:  PR[GP1:91,1] = PR[GP1:90,1] + -61.222;
   1:  PR[GP1:91,2] = PR[GP1:90,2] + 0.261;
   1:L PR[91] 10mm/sec CNT100;
   1:  PR[GP1:91,1] = PR[GP1:90,1] + -60.870;
   1:  PR[GP1:91,2] = PR[GP1:90,2] + -2.903;
   1:L PR[91] 10mm/sec CNT100;
   1:  PR[GP1:91,1] = PR[GP1:90,1] + -59.537;
   1:  PR[GP1:91,2] = PR[GP1:90,2] + -10.698;
   1:L PR[91] 10mm/sec CNT100;
   1:  PR[GP1:91,1] = PR[GP1:90,1] + -58.430;
   1:  PR[GP1:91,2] = PR[GP1:90,2] + -13.748;
   1:L PR[91] 10mm/sec CNT100;
   1:  PR[GP1:91,1] = PR[GP1:90,1] + -54.440;
   1:  PR[GP1:91,2] = PR[GP1:90,2] + -20.973;
   1:L PR[91] 10mm/sec CNT100;
   1:  PR[GP1:91,1] = PR[GP1:90,1] + -52.735;
   1:  PR[GP1:91,2] = PR[GP1:90,2] + -23.635;
   1:L PR[91] 10mm/sec CNT100;
   1:  PR[GP1:91,1] = PR[GP1:90,1] + -50.657;
   1:  PR[GP1:91,2] = PR[GP1:90,2] + -25.673;
   1:L PR[91] 10mm/sec CNT100;
   1:  PR[GP1:91,1] = PR[GP1:90,1] + -44.085;
   1:  PR[GP1:91,2] = PR[GP1:90,2] + -31.635;
   1:L PR[91] 10mm/sec CNT100;
   1:  PR[GP1:91,1] = PR[GP1:90,1] + -41.771;
   1:  PR[GP1:91,2] = PR[GP1:90,2] + -33.094;
   1:L PR[91] 10mm/sec CNT100;
   1:  PR[GP1:91,1] = PR[GP1:90,1] + -32.952;
   1:  PR[GP1:91,2] = PR[GP1:90,2] + -36.975;
   1:L PR[91] 10mm/sec CNT100;
   1:  PR[GP1:91,1] = PR[GP1:90,1] + -30.633;
   1:  PR[GP1:91,2] = PR[GP1:90,2] + -37.825;
   1:L PR[91] 10mm/sec CNT100;
   1:  PR[GP1:91,1] = PR[GP1:90,1] + -28.429;
   1:  PR[GP1:91,2] = PR[GP1:90,2] + -38.138;
   1:L PR[91] 10mm/sec CNT100;
   1:  PR[GP1:91,1] = PR[GP1:90,1] + -18.098;
   1:  PR[GP1:91,2] = PR[GP1:90,2] + -39.130;
   1:L PR[91] 10mm/sec CNT100;
   1:  PR[GP1:91,1] = PR[GP1:90,1] + -16.207;
   1:  PR[GP1:91,2] = PR[GP1:90,2] + -39.005;
   1:L PR[91] 10mm/sec CNT100;
   1:  PR[GP1:91,1] = PR[GP1:90,1] + -5.390;
   1:  PR[GP1:91,2] = PR[GP1:90,2] + -36.530;
   1:L PR[91] 10mm/sec CNT100;
   1:  PR[GP1:91,1] = PR[GP1:90,1] + -3.879;
   1:  PR[GP1:91,2] = PR[GP1:90,2] + -36.096;
   1:L PR[91] 10mm/sec CNT100;
   1:  PR[GP1:91,1] = PR[GP1:90,1] + -0.265;
   1:  PR[GP1:91,2] = PR[GP1:90,2] + -33.979;
   1:L PR[91] 10mm/sec CNT100;
   1:  PR[GP1:91,1] = PR[GP1:90,1] + 3.097;
   1:  PR[GP1:91,2] = PR[GP1:90,2] + -36.165;
   1:  PR[GP1:91,3] = PR[GP1:90,3] + 77.165;
   1:L PR[91] 10mm/sec CNT100;
   1:  PR[GP1:91,1] = PR[GP1:90,1] + 4.489;
   1:  PR[GP1:91,2] = PR[GP1:90,2] + -36.565;
   1:L PR[91] 10mm/sec CNT100;
   1:  PR[GP1:91,1] = PR[GP1:90,1] + 15.504;
   1:  PR[GP1:91,2] = PR[GP1:90,2] + -39.085;
   1:L PR[91] 10mm/sec CNT100;
   1:  PR[GP1:91,1] = PR[GP1:90,1] + 17.254;
   1:  PR[GP1:91,2] = PR[GP1:90,2] + -39.201;
   1:L PR[91] 10mm/sec CNT100;
   1:  PR[GP1:91,1] = PR[GP1:90,1] + 19.260;
   1:  PR[GP1:91,2] = PR[GP1:90,2] + -38.924;
   1:L PR[91] 10mm/sec CNT100;
   1:  PR[GP1:91,1] = PR[GP1:90,1] + 29.889;
   1:  PR[GP1:91,2] = PR[GP1:90,2] + -37.891;
   1:L PR[91] 10mm/sec CNT100;
   1:  PR[GP1:91,1] = PR[GP1:90,1] + 32.072;
   1:  PR[GP1:91,2] = PR[GP1:90,2] + -37.095;
   1:L PR[91] 10mm/sec CNT100;
   1:  PR[GP1:91,1] = PR[GP1:90,1] + 41.091;
   1:  PR[GP1:91,2] = PR[GP1:90,2] + -33.129;
   1:L PR[91] 10mm/sec CNT100;
   1:  PR[GP1:91,1] = PR[GP1:90,1] + 43.271;
   1:  PR[GP1:91,2] = PR[GP1:90,2] + -31.761;
   1:L PR[91] 10mm/sec CNT100;
   1:  PR[GP1:91,1] = PR[GP1:90,1] + 45.278;
   1:  PR[GP1:91,2] = PR[GP1:90,2] + -29.804;
   1:L PR[91] 10mm/sec CNT100;
   1:  PR[GP1:91,1] = PR[GP1:90,1] + 52.001;
   1:  PR[GP1:91,2] = PR[GP1:90,2] + -23.689;
   1:L PR[91] 10mm/sec CNT100;
   1:  PR[GP1:91,1] = PR[GP1:90,1] + 53.644;
   1:  PR[GP1:91,2] = PR[GP1:90,2] + -21.141;
   1:L PR[91] 10mm/sec CNT100;
   1:  PR[GP1:91,1] = PR[GP1:90,1] + 57.741;
   1:  PR[GP1:91,2] = PR[GP1:90,2] + -13.735;
   1:L PR[91] 10mm/sec CNT100;
   1:  PR[GP1:91,1] = PR[GP1:90,1] + 58.792;
   1:  PR[GP1:91,2] = PR[GP1:90,2] + -10.879;
   1:L PR[91] 10mm/sec CNT100;
   1:  PR[GP1:91,1] = PR[GP1:90,1] + 59.149;
   1:  PR[GP1:91,2] = PR[GP1:90,2] + -7.737;
   1:L PR[91] 10mm/sec CNT100;
   1:  PR[GP1:91,1] = PR[GP1:90,1] + 60.519;
   1:  PR[GP1:91,2] = PR[GP1:90,2] + 0.296;
   1:L PR[91] 10mm/sec CNT100;
   1:  PR[GP1:91,1] = PR[GP1:90,1] + 60.168;
   1:  PR[GP1:91,2] = PR[GP1:90,2] + 3.400;
   1:L PR[91] 10mm/sec CNT100;
   1:  PR[GP1:91,1] = PR[GP1:90,1] + 58.792;
   1:  PR[GP1:91,2] = PR[GP1:90,2] + 11.437;
   1:L PR[91] 10mm/sec CNT100;
   1:  PR[GP1:91,1] = PR[GP1:90,1] + 57.735;
   1:  PR[GP1:91,2] = PR[GP1:90,2] + 14.310;
   1:L PR[91] 10mm/sec CNT100;
   1:  PR[GP1:91,1] = PR[GP1:90,1] + 53.620;
   1:  PR[GP1:91,2] = PR[GP1:90,2] + 21.729;
   1:L PR[91] 10mm/sec CNT100;
   1:  PR[GP1:91,1] = PR[GP1:90,1] + 51.971;
   1:  PR[GP1:91,2] = PR[GP1:90,2] + 24.287;
   1:L PR[91] 10mm/sec CNT100;
   1:  PR[GP1:91,1] = PR[GP1:90,1] + 49.987;
   1:  PR[GP1:91,2] = PR[GP1:90,2] + 26.230;
   1:L PR[91] 10mm/sec CNT100;
   1:  PR[GP1:91,1] = PR[GP1:90,1] + 43.229;
   1:  PR[GP1:91,2] = PR[GP1:90,2] + 32.346;
   1:L PR[91] 10mm/sec CNT100;
   1:  PR[GP1:91,1] = PR[GP1:90,1] + 41.040;
   1:  PR[GP1:91,2] = PR[GP1:90,2] + 33.720;
   1:L PR[91] 10mm/sec CNT100;
   1:  PR[GP1:91,1] = PR[GP1:90,1] + 31.987;
   1:  PR[GP1:91,2] = PR[GP1:90,2] + 37.675;
   1:L PR[91] 10mm/sec CNT100;
   1:  PR[GP1:91,1] = PR[GP1:90,1] + 29.791;
   1:  PR[GP1:91,2] = PR[GP1:90,2] + 38.476;
   1:L PR[91] 10mm/sec CNT100;
   1:  PR[GP1:91,1] = PR[GP1:90,1] + 27.715;
   1:  PR[GP1:91,2] = PR[GP1:90,2] + 38.771;
   1:L PR[91] 10mm/sec CNT100;
   1:  PR[GP1:91,1] = PR[GP1:90,1] + 17.148;
   1:  PR[GP1:91,2] = PR[GP1:90,2] + 39.753;
   1:L PR[91] 10mm/sec CNT100;
   1:  PR[GP1:91,1] = PR[GP1:90,1] + 15.388;
   1:  PR[GP1:91,2] = PR[GP1:90,2] + 39.636;
   1:L PR[91] 10mm/sec CNT100;
   1:  PR[GP1:91,1] = PR[GP1:90,1] + 4.193;
   1:  PR[GP1:91,2] = PR[GP1:90,2] + 36.992;
   1:L PR[91] 10mm/sec CNT100;
   1:  PR[GP1:91,1] = PR[GP1:90,1] + 2.881;
   1:  PR[GP1:91,2] = PR[GP1:90,2] + 36.614;
   1:L PR[91] 10mm/sec CNT100;
   1:  PR[GP1:91,1] = PR[GP1:90,1] + 0.882;
   1:  PR[GP1:91,2] = PR[GP1:90,2] + 35.558;
   1:L PR[91] 10mm/sec CNT100;
   1:  PR[GP1:91,1] = PR[GP1:90,1] + -0.263;
   1:  PR[GP1:91,2] = PR[GP1:90,2] + 34.627;
   1:L PR[91] 10mm/sec CNT100;
   1:  PR[GP1:91,1] = PR[GP1:90,1] + -1.406;
   1:  PR[GP1:91,2] = PR[GP1:90,2] + 35.557;
   1:L PR[91] 10mm/sec CNT100;
   1:  PR[GP1:91,1] = PR[GP1:90,1] + -3.404;
   1:  PR[GP1:91,2] = PR[GP1:90,2] + 36.615;
   1:L PR[91] 10mm/sec CNT100;
   1:  PR[GP1:91,1] = PR[GP1:90,1] + -4.714;
   1:  PR[GP1:91,2] = PR[GP1:90,2] + 36.992;
   1:L PR[91] 10mm/sec CNT100;
   1:  PR[GP1:91,1] = PR[GP1:90,1] + -15.913;
   1:  PR[GP1:91,2] = PR[GP1:90,2] + 39.636;
   1:L PR[91] 10mm/sec CNT100;
   1:  PR[GP1:91,1] = PR[GP1:90,1] + -17.665;
   1:  PR[GP1:91,2] = PR[GP1:90,2] + 39.751;
   1:L PR[91] 10mm/sec CNT100;
   1:  PR[GP1:91,1] = PR[GP1:90,1] + -19.678;
   1:  PR[GP1:91,2] = PR[GP1:90,2] + 39.473;
   1:L PR[91] 10mm/sec CNT100;
   1:  PR[GP1:91,1] = PR[GP1:90,1] + -30.342;
   1:  PR[GP1:91,2] = PR[GP1:90,2] + 38.470;
   1:L PR[91] 10mm/sec CNT100;
   1:  PR[GP1:91,1] = PR[GP1:90,1] + -32.522;
   1:  PR[GP1:91,2] = PR[GP1:90,2] + 37.672;
   1:L PR[91] 10mm/sec CNT100;
   1:  PR[GP1:91,1] = PR[GP1:90,1] + -41.575;
   1:  PR[GP1:91,2] = PR[GP1:90,2] + 33.714;
   1:L PR[91] 10mm/sec CNT100;
   1:  PR[GP1:91,1] = PR[GP1:90,1] + -43.767;
   1:  PR[GP1:91,2] = PR[GP1:90,2] + 32.331;
   1:L PR[91] 10mm/sec CNT100;
   1:  PR[GP1:91,1] = PR[GP1:90,1] + -45.780;
   1:  PR[GP1:91,2] = PR[GP1:90,2] + 30.367;
   1:L PR[91] 10mm/sec CNT100;
   1:  PR[GP1:91,1] = PR[GP1:90,1] + -52.530;
   1:  PR[GP1:91,2] = PR[GP1:90,2] + 24.255;
   1:L PR[91] 10mm/sec CNT100;
   1:  PR[GP1:91,1] = PR[GP1:90,1] + -54.155;
   1:  PR[GP1:91,2] = PR[GP1:90,2] + 21.719;
   1:L PR[91] 10mm/sec CNT100;
   1:  PR[GP1:91,1] = PR[GP1:90,1] + -58.269;
   1:  PR[GP1:91,2] = PR[GP1:90,2] + 14.287;
   1:L PR[91] 10mm/sec CNT100;
   1:  PR[GP1:91,1] = PR[GP1:90,1] + -59.325;
   1:  PR[GP1:91,2] = PR[GP1:90,2] + 11.379;
   1:L PR[91] 10mm/sec CNT100;
   1:  PR[GP1:91,1] = PR[GP1:90,1] + -59.669;
   1:  PR[GP1:91,2] = PR[GP1:90,2] + 8.303;
   1:L PR[91] 10mm/sec CNT100;
   1:  PR[GP1:91,1] = PR[GP1:90,1] + -61.045;
   1:  PR[GP1:91,2] = PR[GP1:90,2] + 0.261;
   1:L PR[91] 10mm/sec CNT100;
   1:  PR[GP1:91,1] = PR[GP1:90,1] + -60.707;
   1:  PR[GP1:91,2] = PR[GP1:90,2] + -2.775;
   1:L PR[91] 10mm/sec CNT100;
   1:  PR[GP1:91,1] = PR[GP1:90,1] + -59.337;
   1:  PR[GP1:91,2] = PR[GP1:90,2] + -10.788;
   1:L PR[91] 10mm/sec CNT100;
   1:  PR[GP1:91,1] = PR[GP1:90,1] + -58.275;
   1:  PR[GP1:91,2] = PR[GP1:90,2] + -13.712;
   1:L PR[91] 10mm/sec CNT100;
   1:  PR[GP1:91,1] = PR[GP1:90,1] + -54.178;
   1:  PR[GP1:91,2] = PR[GP1:90,2] + -21.131;
   1:L PR[91] 10mm/sec CNT100;
   1:  PR[GP1:91,1] = PR[GP1:90,1] + -52.547;
   1:  PR[GP1:91,2] = PR[GP1:90,2] + -23.677;
   1:L PR[91] 10mm/sec CNT100;
   1:  PR[GP1:91,1] = PR[GP1:90,1] + -50.560;
   1:  PR[GP1:91,2] = PR[GP1:90,2] + -25.627;
   1:L PR[91] 10mm/sec CNT100;
   1:  PR[GP1:91,1] = PR[GP1:90,1] + -43.829;
   1:  PR[GP1:91,2] = PR[GP1:90,2] + -31.733;
   1:L PR[91] 10mm/sec CNT100;
   1:  PR[GP1:91,1] = PR[GP1:90,1] + -41.626;
   1:  PR[GP1:91,2] = PR[GP1:90,2] + -33.122;
   1:L PR[91] 10mm/sec CNT100;
   1:  PR[GP1:91,1] = PR[GP1:90,1] + -32.608;
   1:  PR[GP1:91,2] = PR[GP1:90,2] + -37.091;
   1:L PR[91] 10mm/sec CNT100;
   1:  PR[GP1:91,1] = PR[GP1:90,1] + -30.415;
   1:  PR[GP1:91,2] = PR[GP1:90,2] + -37.894;
   1:L PR[91] 10mm/sec CNT100;
   1:  PR[GP1:91,1] = PR[GP1:90,1] + -28.331;
   1:  PR[GP1:91,2] = PR[GP1:90,2] + -38.191;
   1:L PR[91] 10mm/sec CNT100;
   1:  PR[GP1:91,1] = PR[GP1:90,1] + -17.798;
   1:  PR[GP1:91,2] = PR[GP1:90,2] + -39.202;
   1:L PR[91] 10mm/sec CNT100;
   1:  PR[GP1:91,1] = PR[GP1:90,1] + -16.030;
   1:  PR[GP1:91,2] = PR[GP1:90,2] + -39.085;
   1:L PR[91] 10mm/sec CNT100;
   1:  PR[GP1:91,1] = PR[GP1:90,1] + -5.015;
   1:  PR[GP1:91,2] = PR[GP1:90,2] + -36.565;
   1:L PR[91] 10mm/sec CNT100;
   1:  PR[GP1:91,1] = PR[GP1:90,1] + -3.625;
   1:  PR[GP1:91,2] = PR[GP1:90,2] + -36.166;
   1:L PR[91] 10mm/sec CNT100;
   1:  PR[GP1:91,1] = PR[GP1:90,1] + -0.265;
   1:  PR[GP1:91,2] = PR[GP1:90,2] + -34.197;
   1:L PR[91] 10mm/sec CNT100;
   1:  PR[GP1:91,1] = PR[GP1:90,1] + 2.842;
   1:  PR[GP1:91,2] = PR[GP1:90,2] + -36.234;
   1:  PR[GP1:91,3] = PR[GP1:90,3] + 77.775;
   1:L PR[91] 10mm/sec CNT100;
   1:  PR[GP1:91,1] = PR[GP1:90,1] + 4.113;
   1:  PR[GP1:91,2] = PR[GP1:90,2] + -36.599;
   1:L PR[91] 10mm/sec CNT100;
   1:  PR[GP1:91,1] = PR[GP1:90,1] + 15.327;
   1:  PR[GP1:91,2] = PR[GP1:90,2] + -39.165;
   1:L PR[91] 10mm/sec CNT100;
   1:  PR[GP1:91,1] = PR[GP1:90,1] + 16.954;
   1:  PR[GP1:91,2] = PR[GP1:90,2] + -39.273;
   1:L PR[91] 10mm/sec CNT100;
   1:  PR[GP1:91,1] = PR[GP1:90,1] + 18.824;
   1:  PR[GP1:91,2] = PR[GP1:90,2] + -39.015;
   1:L PR[91] 10mm/sec CNT100;
   1:  PR[GP1:91,1] = PR[GP1:90,1] + 29.672;
   1:  PR[GP1:91,2] = PR[GP1:90,2] + -37.961;
   1:L PR[91] 10mm/sec CNT100;
   1:  PR[GP1:91,1] = PR[GP1:90,1] + 31.728;
   1:  PR[GP1:91,2] = PR[GP1:90,2] + -37.210;
   1:L PR[91] 10mm/sec CNT100;
   1:  PR[GP1:91,1] = PR[GP1:90,1] + 40.946;
   1:  PR[GP1:91,2] = PR[GP1:90,2] + -33.157;
   1:L PR[91] 10mm/sec CNT100;
   1:  PR[GP1:91,1] = PR[GP1:90,1] + 43.015;
   1:  PR[GP1:91,2] = PR[GP1:90,2] + -31.859;
   1:L PR[91] 10mm/sec CNT100;
   1:  PR[GP1:91,1] = PR[GP1:90,1] + 44.923;
   1:  PR[GP1:91,2] = PR[GP1:90,2] + -29.999;
   1:L PR[91] 10mm/sec CNT100;
   1:  PR[GP1:91,1] = PR[GP1:90,1] + 51.814;
   1:  PR[GP1:91,2] = PR[GP1:90,2] + -23.731;
   1:L PR[91] 10mm/sec CNT100;
   1:  PR[GP1:91,1] = PR[GP1:90,1] + 53.382;
   1:  PR[GP1:91,2] = PR[GP1:90,2] + -21.299;
   1:L PR[91] 10mm/sec CNT100;
   1:  PR[GP1:91,1] = PR[GP1:90,1] + 57.587;
   1:  PR[GP1:91,2] = PR[GP1:90,2] + -13.698;
   1:L PR[91] 10mm/sec CNT100;
   1:  PR[GP1:91,1] = PR[GP1:90,1] + 58.592;
   1:  PR[GP1:91,2] = PR[GP1:90,2] + -10.965;
   1:L PR[91] 10mm/sec CNT100;
   1:  PR[GP1:91,1] = PR[GP1:90,1] + 58.934;
   1:  PR[GP1:91,2] = PR[GP1:90,2] + -7.956;
   1:L PR[91] 10mm/sec CNT100;
   1:  PR[GP1:91,1] = PR[GP1:90,1] + 60.342;
   1:  PR[GP1:91,2] = PR[GP1:90,2] + 0.296;
   1:L PR[91] 10mm/sec CNT100;
   1:  PR[GP1:91,1] = PR[GP1:90,1] + 60.005;
   1:  PR[GP1:91,2] = PR[GP1:90,2] + 3.269;
   1:L PR[91] 10mm/sec CNT100;
   1:  PR[GP1:91,1] = PR[GP1:90,1] + 58.592;
   1:  PR[GP1:91,2] = PR[GP1:90,2] + 11.524;
   1:L PR[91] 10mm/sec CNT100;
   1:  PR[GP1:91,1] = PR[GP1:90,1] + 57.581;
   1:  PR[GP1:91,2] = PR[GP1:90,2] + 14.273;
   1:L PR[91] 10mm/sec CNT100;
   1:  PR[GP1:91,1] = PR[GP1:90,1] + 53.358;
   1:  PR[GP1:91,2] = PR[GP1:90,2] + 21.887;
   1:L PR[91] 10mm/sec CNT100;
   1:  PR[GP1:91,1] = PR[GP1:90,1] + 51.784;
   1:  PR[GP1:91,2] = PR[GP1:90,2] + 24.329;
   1:L PR[91] 10mm/sec CNT100;
   1:  PR[GP1:91,1] = PR[GP1:90,1] + 49.890;
   1:  PR[GP1:91,2] = PR[GP1:90,2] + 26.184;
   1:L PR[91] 10mm/sec CNT100;
   1:  PR[GP1:91,1] = PR[GP1:90,1] + 42.972;
   1:  PR[GP1:91,2] = PR[GP1:90,2] + 32.445;
   1:L PR[91] 10mm/sec CNT100;
   1:  PR[GP1:91,1] = PR[GP1:90,1] + 40.893;
   1:  PR[GP1:91,2] = PR[GP1:90,2] + 33.749;
   1:L PR[91] 10mm/sec CNT100;
   1:  PR[GP1:91,1] = PR[GP1:90,1] + 31.641;
   1:  PR[GP1:91,2] = PR[GP1:90,2] + 37.791;
   1:L PR[91] 10mm/sec CNT100;
   1:  PR[GP1:91,1] = PR[GP1:90,1] + 29.572;
   1:  PR[GP1:91,2] = PR[GP1:90,2] + 38.546;
   1:L PR[91] 10mm/sec CNT100;
   1:  PR[GP1:91,1] = PR[GP1:90,1] + 27.616;
   1:  PR[GP1:91,2] = PR[GP1:90,2] + 38.824;
   1:L PR[91] 10mm/sec CNT100;
   1:  PR[GP1:91,1] = PR[GP1:90,1] + 16.846;
   1:  PR[GP1:91,2] = PR[GP1:90,2] + 39.825;
   1:L PR[91] 10mm/sec CNT100;
   1:  PR[GP1:91,1] = PR[GP1:90,1] + 15.209;
   1:  PR[GP1:91,2] = PR[GP1:90,2] + 39.716;
   1:L PR[91] 10mm/sec CNT100;
   1:  PR[GP1:91,1] = PR[GP1:90,1] + 3.812;
   1:  PR[GP1:91,2] = PR[GP1:90,2] + 37.024;
   1:L PR[91] 10mm/sec CNT100;
   1:  PR[GP1:91,1] = PR[GP1:90,1] + 2.622;
   1:  PR[GP1:91,2] = PR[GP1:90,2] + 36.682;
   1:L PR[91] 10mm/sec CNT100;
   1:  PR[GP1:91,1] = PR[GP1:90,1] + 0.709;
   1:  PR[GP1:91,2] = PR[GP1:90,2] + 35.672;
   1:L PR[91] 10mm/sec CNT100;
   1:  PR[GP1:91,1] = PR[GP1:90,1] + -0.263;
   1:  PR[GP1:91,2] = PR[GP1:90,2] + 34.882;
   1:L PR[91] 10mm/sec CNT100;
   1:  PR[GP1:91,1] = PR[GP1:90,1] + -1.234;
   1:  PR[GP1:91,2] = PR[GP1:90,2] + 35.671;
   1:L PR[91] 10mm/sec CNT100;
   1:  PR[GP1:91,1] = PR[GP1:90,1] + -3.146;
   1:  PR[GP1:91,2] = PR[GP1:90,2] + 36.683;
   1:L PR[91] 10mm/sec CNT100;
   1:  PR[GP1:91,1] = PR[GP1:90,1] + -4.334;
   1:  PR[GP1:91,2] = PR[GP1:90,2] + 37.024;
   1:L PR[91] 10mm/sec CNT100;
   1:  PR[GP1:91,1] = PR[GP1:90,1] + -15.734;
   1:  PR[GP1:91,2] = PR[GP1:90,2] + 39.716;
   1:L PR[91] 10mm/sec CNT100;
   1:  PR[GP1:91,1] = PR[GP1:90,1] + -17.363;
   1:  PR[GP1:91,2] = PR[GP1:90,2] + 39.823;
   1:L PR[91] 10mm/sec CNT100;
   1:  PR[GP1:91,1] = PR[GP1:90,1] + -19.238;
   1:  PR[GP1:91,2] = PR[GP1:90,2] + 39.563;
   1:L PR[91] 10mm/sec CNT100;
   1:  PR[GP1:91,1] = PR[GP1:90,1] + -30.122;
   1:  PR[GP1:91,2] = PR[GP1:90,2] + 38.540;
   1:L PR[91] 10mm/sec CNT100;
   1:  PR[GP1:91,1] = PR[GP1:90,1] + -32.175;
   1:  PR[GP1:91,2] = PR[GP1:90,2] + 37.788;
   1:L PR[91] 10mm/sec CNT100;
   1:  PR[GP1:91,1] = PR[GP1:90,1] + -41.428;
   1:  PR[GP1:91,2] = PR[GP1:90,2] + 33.743;
   1:L PR[91] 10mm/sec CNT100;
   1:  PR[GP1:91,1] = PR[GP1:90,1] + -43.510;
   1:  PR[GP1:91,2] = PR[GP1:90,2] + 32.430;
   1:L PR[91] 10mm/sec CNT100;
   1:  PR[GP1:91,1] = PR[GP1:90,1] + -45.422;
   1:  PR[GP1:91,2] = PR[GP1:90,2] + 30.563;
   1:L PR[91] 10mm/sec CNT100;
   1:  PR[GP1:91,1] = PR[GP1:90,1] + -52.341;
   1:  PR[GP1:91,2] = PR[GP1:90,2] + 24.299;
   1:L PR[91] 10mm/sec CNT100;
   1:  PR[GP1:91,1] = PR[GP1:90,1] + -53.892;
   1:  PR[GP1:91,2] = PR[GP1:90,2] + 21.878;
   1:L PR[91] 10mm/sec CNT100;
   1:  PR[GP1:91,1] = PR[GP1:90,1] + -58.115;
   1:  PR[GP1:91,2] = PR[GP1:90,2] + 14.251;
   1:L PR[91] 10mm/sec CNT100;
   1:  PR[GP1:91,1] = PR[GP1:90,1] + -59.124;
   1:  PR[GP1:91,2] = PR[GP1:90,2] + 11.469;
   1:L PR[91] 10mm/sec CNT100;
   1:  PR[GP1:91,1] = PR[GP1:90,1] + -59.454;
   1:  PR[GP1:91,2] = PR[GP1:90,2] + 8.523;
   1:L PR[91] 10mm/sec CNT100;
   1:  PR[GP1:91,1] = PR[GP1:90,1] + -60.868;
   1:  PR[GP1:91,2] = PR[GP1:90,2] + 0.261;
   1:L PR[91] 10mm/sec CNT100;
   1:  PR[GP1:91,1] = PR[GP1:90,1] + -60.544;
   1:  PR[GP1:91,2] = PR[GP1:90,2] + -2.647;
   1:L PR[91] 10mm/sec CNT100;
   1:  PR[GP1:91,1] = PR[GP1:90,1] + -59.136;
   1:  PR[GP1:91,2] = PR[GP1:90,2] + -10.877;
   1:L PR[91] 10mm/sec CNT100;
   1:  PR[GP1:91,1] = PR[GP1:90,1] + -58.121;
   1:  PR[GP1:91,2] = PR[GP1:90,2] + -13.676;
   1:L PR[91] 10mm/sec CNT100;
   1:  PR[GP1:91,1] = PR[GP1:90,1] + -53.916;
   1:  PR[GP1:91,2] = PR[GP1:90,2] + -21.290;
   1:L PR[91] 10mm/sec CNT100;
   1:  PR[GP1:91,1] = PR[GP1:90,1] + -52.359;
   1:  PR[GP1:91,2] = PR[GP1:90,2] + -23.720;
   1:L PR[91] 10mm/sec CNT100;
   1:  PR[GP1:91,1] = PR[GP1:90,1] + -50.462;
   1:  PR[GP1:91,2] = PR[GP1:90,2] + -25.581;
   1:L PR[91] 10mm/sec CNT100;
   1:  PR[GP1:91,1] = PR[GP1:90,1] + -43.572;
   1:  PR[GP1:91,2] = PR[GP1:90,2] + -31.832;
   1:L PR[91] 10mm/sec CNT100;
   1:  PR[GP1:91,1] = PR[GP1:90,1] + -41.480;
   1:  PR[GP1:91,2] = PR[GP1:90,2] + -33.151;
   1:L PR[91] 10mm/sec CNT100;
   1:  PR[GP1:91,1] = PR[GP1:90,1] + -32.263;
   1:  PR[GP1:91,2] = PR[GP1:90,2] + -37.207;
   1:L PR[91] 10mm/sec CNT100;
   1:  PR[GP1:91,1] = PR[GP1:90,1] + -30.197;
   1:  PR[GP1:91,2] = PR[GP1:90,2] + -37.964;
   1:L PR[91] 10mm/sec CNT100;
   1:  PR[GP1:91,1] = PR[GP1:90,1] + -28.233;
   1:  PR[GP1:91,2] = PR[GP1:90,2] + -38.244;
   1:L PR[91] 10mm/sec CNT100;
   1:  PR[GP1:91,1] = PR[GP1:90,1] + -17.497;
   1:  PR[GP1:91,2] = PR[GP1:90,2] + -39.274;
   1:L PR[91] 10mm/sec CNT100;
   1:  PR[GP1:91,1] = PR[GP1:90,1] + -15.853;
   1:  PR[GP1:91,2] = PR[GP1:90,2] + -39.165;
   1:L PR[91] 10mm/sec CNT100;
   1:  PR[GP1:91,1] = PR[GP1:90,1] + -4.639;
   1:  PR[GP1:91,2] = PR[GP1:90,2] + -36.600;
   1:L PR[91] 10mm/sec CNT100;
   1:  PR[GP1:91,1] = PR[GP1:90,1] + -3.370;
   1:  PR[GP1:91,2] = PR[GP1:90,2] + -36.235;
   1:L PR[91] 10mm/sec CNT100;
   1:  PR[GP1:91,1] = PR[GP1:90,1] + -0.265;
   1:  PR[GP1:91,2] = PR[GP1:90,2] + -34.416;
   1:L PR[91] 10mm/sec CNT100;
   1:  PR[GP1:91,1] = PR[GP1:90,1] + 2.587;
   1:  PR[GP1:91,2] = PR[GP1:90,2] + -36.304;
   1:  PR[GP1:91,3] = PR[GP1:90,3] + 78.385;
   1:L PR[91] 10mm/sec CNT100;
   1:  PR[GP1:91,1] = PR[GP1:90,1] + 3.738;
   1:  PR[GP1:91,2] = PR[GP1:90,2] + -36.634;
   1:L PR[91] 10mm/sec CNT100;
   1:  PR[GP1:91,1] = PR[GP1:90,1] + 15.150;
   1:  PR[GP1:91,2] = PR[GP1:90,2] + -39.245;
   1:L PR[91] 10mm/sec CNT100;
   1:  PR[GP1:91,1] = PR[GP1:90,1] + 16.654;
   1:  PR[GP1:91,2] = PR[GP1:90,2] + -39.345;
   1:L PR[91] 10mm/sec CNT100;
   1:  PR[GP1:91,1] = PR[GP1:90,1] + 18.388;
   1:  PR[GP1:91,2] = PR[GP1:90,2] + -39.106;
   1:L PR[91] 10mm/sec CNT100;
   1:  PR[GP1:91,1] = PR[GP1:90,1] + 29.454;
   1:  PR[GP1:91,2] = PR[GP1:90,2] + -38.031;
   1:L PR[91] 10mm/sec CNT100;
   1:  PR[GP1:91,1] = PR[GP1:90,1] + 31.384;
   1:  PR[GP1:91,2] = PR[GP1:90,2] + -37.326;
   1:L PR[91] 10mm/sec CNT100;
   1:  PR[GP1:91,1] = PR[GP1:90,1] + 40.800;
   1:  PR[GP1:91,2] = PR[GP1:90,2] + -33.185;
   1:L PR[91] 10mm/sec CNT100;
   1:  PR[GP1:91,1] = PR[GP1:90,1] + 42.760;
   1:  PR[GP1:91,2] = PR[GP1:90,2] + -31.956;
   1:L PR[91] 10mm/sec CNT100;
   1:  PR[GP1:91,1] = PR[GP1:90,1] + 44.568;
   1:  PR[GP1:91,2] = PR[GP1:90,2] + -30.193;
   1:L PR[91] 10mm/sec CNT100;
   1:  PR[GP1:91,1] = PR[GP1:90,1] + 51.627;
   1:  PR[GP1:91,2] = PR[GP1:90,2] + -23.773;
   1:L PR[91] 10mm/sec CNT100;
   1:  PR[GP1:91,1] = PR[GP1:90,1] + 53.120;
   1:  PR[GP1:91,2] = PR[GP1:90,2] + -21.456;
   1:L PR[91] 10mm/sec CNT100;
   1:  PR[GP1:91,1] = PR[GP1:90,1] + 57.433;
   1:  PR[GP1:91,2] = PR[GP1:90,2] + -13.662;
   1:L PR[91] 10mm/sec CNT100;
   1:  PR[GP1:91,1] = PR[GP1:90,1] + 58.392;
   1:  PR[GP1:91,2] = PR[GP1:90,2] + -11.052;
   1:L PR[91] 10mm/sec CNT100;
   1:  PR[GP1:91,1] = PR[GP1:90,1] + 58.719;
   1:  PR[GP1:91,2] = PR[GP1:90,2] + -8.176;
   1:L PR[91] 10mm/sec CNT100;
   1:  PR[GP1:91,1] = PR[GP1:90,1] + 60.164;
   1:  PR[GP1:91,2] = PR[GP1:90,2] + 0.296;
   1:L PR[91] 10mm/sec CNT100;
   1:  PR[GP1:91,1] = PR[GP1:90,1] + 59.843;
   1:  PR[GP1:91,2] = PR[GP1:90,2] + 3.138;
   1:L PR[91] 10mm/sec CNT100;
   1:  PR[GP1:91,1] = PR[GP1:90,1] + 58.392;
   1:  PR[GP1:91,2] = PR[GP1:90,2] + 11.612;
   1:L PR[91] 10mm/sec CNT100;
   1:  PR[GP1:91,1] = PR[GP1:90,1] + 57.427;
   1:  PR[GP1:91,2] = PR[GP1:90,2] + 14.237;
   1:L PR[91] 10mm/sec CNT100;
   1:  PR[GP1:91,1] = PR[GP1:90,1] + 53.096;
   1:  PR[GP1:91,2] = PR[GP1:90,2] + 22.046;
   1:L PR[91] 10mm/sec CNT100;
   1:  PR[GP1:91,1] = PR[GP1:90,1] + 51.596;
   1:  PR[GP1:91,2] = PR[GP1:90,2] + 24.371;
   1:L PR[91] 10mm/sec CNT100;
   1:  PR[GP1:91,1] = PR[GP1:90,1] + 49.792;
   1:  PR[GP1:91,2] = PR[GP1:90,2] + 26.138;
   1:L PR[91] 10mm/sec CNT100;
   1:  PR[GP1:91,1] = PR[GP1:90,1] + 42.715;
   1:  PR[GP1:91,2] = PR[GP1:90,2] + 32.543;
   1:L PR[91] 10mm/sec CNT100;
   1:  PR[GP1:91,1] = PR[GP1:90,1] + 40.747;
   1:  PR[GP1:91,2] = PR[GP1:90,2] + 33.778;
   1:L PR[91] 10mm/sec CNT100;
   1:  PR[GP1:91,1] = PR[GP1:90,1] + 31.295;
   1:  PR[GP1:91,2] = PR[GP1:90,2] + 37.908;
   1:L PR[91] 10mm/sec CNT100;
   1:  PR[GP1:91,1] = PR[GP1:90,1] + 29.353;
   1:  PR[GP1:91,2] = PR[GP1:90,2] + 38.617;
   1:L PR[91] 10mm/sec CNT100;
   1:  PR[GP1:91,1] = PR[GP1:90,1] + 27.517;
   1:  PR[GP1:91,2] = PR[GP1:90,2] + 38.877;
   1:L PR[91] 10mm/sec CNT100;
   1:  PR[GP1:91,1] = PR[GP1:90,1] + 16.544;
   1:  PR[GP1:91,2] = PR[GP1:90,2] + 39.896;
   1:L PR[91] 10mm/sec CNT100;
   1:  PR[GP1:91,1] = PR[GP1:90,1] + 15.031;
   1:  PR[GP1:91,2] = PR[GP1:90,2] + 39.796;
   1:L PR[91] 10mm/sec CNT100;
   1:  PR[GP1:91,1] = PR[GP1:90,1] + 3.431;
   1:  PR[GP1:91,2] = PR[GP1:90,2] + 37.056;
   1:L PR[91] 10mm/sec CNT100;
   1:  PR[GP1:91,1] = PR[GP1:90,1] + 2.364;
   1:  PR[GP1:91,2] = PR[GP1:90,2] + 36.750;
   1:L PR[91] 10mm/sec CNT100;
   1:  PR[GP1:91,1] = PR[GP1:90,1] + 0.536;
   1:  PR[GP1:91,2] = PR[GP1:90,2] + 35.786;
   1:L PR[91] 10mm/sec CNT100;
   1:  PR[GP1:91,1] = PR[GP1:90,1] + -0.263;
   1:  PR[GP1:91,2] = PR[GP1:90,2] + 35.137;
   1:L PR[91] 10mm/sec CNT100;
   1:  PR[GP1:91,1] = PR[GP1:90,1] + -1.061;
   1:  PR[GP1:91,2] = PR[GP1:90,2] + 35.785;
   1:L PR[91] 10mm/sec CNT100;
   1:  PR[GP1:91,1] = PR[GP1:90,1] + -2.888;
   1:  PR[GP1:91,2] = PR[GP1:90,2] + 36.750;
   1:L PR[91] 10mm/sec CNT100;
   1:  PR[GP1:91,1] = PR[GP1:90,1] + -3.953;
   1:  PR[GP1:91,2] = PR[GP1:90,2] + 37.057;
   1:L PR[91] 10mm/sec CNT100;
   1:  PR[GP1:91,1] = PR[GP1:90,1] + -15.556;
   1:  PR[GP1:91,2] = PR[GP1:90,2] + 39.796;
   1:L PR[91] 10mm/sec CNT100;
   1:  PR[GP1:91,1] = PR[GP1:90,1] + -17.060;
   1:  PR[GP1:91,2] = PR[GP1:90,2] + 39.895;
   1:L PR[91] 10mm/sec CNT100;
   1:  PR[GP1:91,1] = PR[GP1:90,1] + -18.799;
   1:  PR[GP1:91,2] = PR[GP1:90,2] + 39.654;
   1:L PR[91] 10mm/sec CNT100;
   1:  PR[GP1:91,1] = PR[GP1:90,1] + -29.902;
   1:  PR[GP1:91,2] = PR[GP1:90,2] + 38.610;
   1:L PR[91] 10mm/sec CNT100;
   1:  PR[GP1:91,1] = PR[GP1:90,1] + -31.829;
   1:  PR[GP1:91,2] = PR[GP1:90,2] + 37.905;
   1:L PR[91] 10mm/sec CNT100;
   1:  PR[GP1:91,1] = PR[GP1:90,1] + -41.281;
   1:  PR[GP1:91,2] = PR[GP1:90,2] + 33.772;
   1:L PR[91] 10mm/sec CNT100;
   1:  PR[GP1:91,1] = PR[GP1:90,1] + -43.252;
   1:  PR[GP1:91,2] = PR[GP1:90,2] + 32.530;
   1:L PR[91] 10mm/sec CNT100;
   1:  PR[GP1:91,1] = PR[GP1:90,1] + -45.064;
   1:  PR[GP1:91,2] = PR[GP1:90,2] + 30.760;
   1:L PR[91] 10mm/sec CNT100;
   1:  PR[GP1:91,1] = PR[GP1:90,1] + -52.152;
   1:  PR[GP1:91,2] = PR[GP1:90,2] + 24.342;
   1:L PR[91] 10mm/sec CNT100;
   1:  PR[GP1:91,1] = PR[GP1:90,1] + -53.629;
   1:  PR[GP1:91,2] = PR[GP1:90,2] + 22.037;
   1:L PR[91] 10mm/sec CNT100;
   1:  PR[GP1:91,1] = PR[GP1:90,1] + -57.960;
   1:  PR[GP1:91,2] = PR[GP1:90,2] + 14.215;
   1:L PR[91] 10mm/sec CNT100;
   1:  PR[GP1:91,1] = PR[GP1:90,1] + -58.924;
   1:  PR[GP1:91,2] = PR[GP1:90,2] + 11.559;
   1:L PR[91] 10mm/sec CNT100;
   1:  PR[GP1:91,1] = PR[GP1:90,1] + -59.239;
   1:  PR[GP1:91,2] = PR[GP1:90,2] + 8.743;
   1:L PR[91] 10mm/sec CNT100;
   1:  PR[GP1:91,1] = PR[GP1:90,1] + -60.691;
   1:  PR[GP1:91,2] = PR[GP1:90,2] + 0.261;
   1:L PR[91] 10mm/sec CNT100;
   1:  PR[GP1:91,1] = PR[GP1:90,1] + -60.381;
   1:  PR[GP1:91,2] = PR[GP1:90,2] + -2.519;
   1:L PR[91] 10mm/sec CNT100;
   1:  PR[GP1:91,1] = PR[GP1:90,1] + -58.936;
   1:  PR[GP1:91,2] = PR[GP1:90,2] + -10.966;
   1:L PR[91] 10mm/sec CNT100;
   1:  PR[GP1:91,1] = PR[GP1:90,1] + -57.966;
   1:  PR[GP1:91,2] = PR[GP1:90,2] + -13.639;
   1:L PR[91] 10mm/sec CNT100;
   1:  PR[GP1:91,1] = PR[GP1:90,1] + -53.654;
   1:  PR[GP1:91,2] = PR[GP1:90,2] + -21.448;
   1:L PR[91] 10mm/sec CNT100;
   1:  PR[GP1:91,1] = PR[GP1:90,1] + -52.171;
   1:  PR[GP1:91,2] = PR[GP1:90,2] + -23.763;
   1:L PR[91] 10mm/sec CNT100;
   1:  PR[GP1:91,1] = PR[GP1:90,1] + -50.364;
   1:  PR[GP1:91,2] = PR[GP1:90,2] + -25.536;
   1:L PR[91] 10mm/sec CNT100;
   1:  PR[GP1:91,1] = PR[GP1:90,1] + -43.315;
   1:  PR[GP1:91,2] = PR[GP1:90,2] + -31.930;
   1:L PR[91] 10mm/sec CNT100;
   1:  PR[GP1:91,1] = PR[GP1:90,1] + -41.335;
   1:  PR[GP1:91,2] = PR[GP1:90,2] + -33.179;
   1:L PR[91] 10mm/sec CNT100;
   1:  PR[GP1:91,1] = PR[GP1:90,1] + -31.919;
   1:  PR[GP1:91,2] = PR[GP1:90,2] + -37.323;
   1:L PR[91] 10mm/sec CNT100;
   1:  PR[GP1:91,1] = PR[GP1:90,1] + -29.978;
   1:  PR[GP1:91,2] = PR[GP1:90,2] + -38.034;
   1:L PR[91] 10mm/sec CNT100;
   1:  PR[GP1:91,1] = PR[GP1:90,1] + -28.135;
   1:  PR[GP1:91,2] = PR[GP1:90,2] + -38.296;
   1:L PR[91] 10mm/sec CNT100;
   1:  PR[GP1:91,1] = PR[GP1:90,1] + -17.197;
   1:  PR[GP1:91,2] = PR[GP1:90,2] + -39.346;
   1:L PR[91] 10mm/sec CNT100;
   1:  PR[GP1:91,1] = PR[GP1:90,1] + -15.676;
   1:  PR[GP1:91,2] = PR[GP1:90,2] + -39.245;
   1:L PR[91] 10mm/sec CNT100;
   1:  PR[GP1:91,1] = PR[GP1:90,1] + -4.264;
   1:  PR[GP1:91,2] = PR[GP1:90,2] + -36.634;
   1:L PR[91] 10mm/sec CNT100;
   1:  PR[GP1:91,1] = PR[GP1:90,1] + -3.115;
   1:  PR[GP1:91,2] = PR[GP1:90,2] + -36.304;
   1:L PR[91] 10mm/sec CNT100;
   1:  PR[GP1:91,1] = PR[GP1:90,1] + -0.265;
   1:  PR[GP1:91,2] = PR[GP1:90,2] + -34.634;
   1:L PR[91] 10mm/sec CNT100;
   1:  PR[GP1:91,1] = PR[GP1:90,1] + 2.333;
   1:  PR[GP1:91,2] = PR[GP1:90,2] + -36.373;
   1:  PR[GP1:91,3] = PR[GP1:90,3] + 78.995;
   1:L PR[91] 10mm/sec CNT100;
   1:  PR[GP1:91,1] = PR[GP1:90,1] + 3.363;
   1:  PR[GP1:91,2] = PR[GP1:90,2] + -36.669;
   1:L PR[91] 10mm/sec CNT100;
   1:  PR[GP1:91,1] = PR[GP1:90,1] + 14.974;
   1:  PR[GP1:91,2] = PR[GP1:90,2] + -39.326;
   1:L PR[91] 10mm/sec CNT100;
   1:  PR[GP1:91,1] = PR[GP1:90,1] + 16.354;
   1:  PR[GP1:91,2] = PR[GP1:90,2] + -39.417;
   1:L PR[91] 10mm/sec CNT100;
   1:  PR[GP1:91,1] = PR[GP1:90,1] + 17.952;
   1:  PR[GP1:91,2] = PR[GP1:90,2] + -39.197;
   1:L PR[91] 10mm/sec CNT100;
   1:  PR[GP1:91,1] = PR[GP1:90,1] + 29.237;
   1:  PR[GP1:91,2] = PR[GP1:90,2] + -38.100;
   1:L PR[91] 10mm/sec CNT100;
   1:  PR[GP1:91,1] = PR[GP1:90,1] + 31.040;
   1:  PR[GP1:91,2] = PR[GP1:90,2] + -37.442;
   1:L PR[91] 10mm/sec CNT100;
   1:  PR[GP1:91,1] = PR[GP1:90,1] + 40.655;
   1:  PR[GP1:91,2] = PR[GP1:90,2] + -33.214;
   1:L PR[91] 10mm/sec CNT100;
   1:  PR[GP1:91,1] = PR[GP1:90,1] + 42.504;
   1:  PR[GP1:91,2] = PR[GP1:90,2] + -32.054;
   1:L PR[91] 10mm/sec CNT100;
   1:  PR[GP1:91,1] = PR[GP1:90,1] + 44.213;
   1:  PR[GP1:91,2] = PR[GP1:90,2] + -30.388;
   1:L PR[91] 10mm/sec CNT100;
   1:  PR[GP1:91,1] = PR[GP1:90,1] + 51.440;
   1:  PR[GP1:91,2] = PR[GP1:90,2] + -23.814;
   1:L PR[91] 10mm/sec CNT100;
   1:  PR[GP1:91,1] = PR[GP1:90,1] + 52.859;
   1:  PR[GP1:91,2] = PR[GP1:90,2] + -21.614;
   1:L PR[91] 10mm/sec CNT100;
   1:  PR[GP1:91,1] = PR[GP1:90,1] + 57.279;
   1:  PR[GP1:91,2] = PR[GP1:90,2] + -13.625;
   1:L PR[91] 10mm/sec CNT100;
   1:  PR[GP1:91,1] = PR[GP1:90,1] + 58.193;
   1:  PR[GP1:91,2] = PR[GP1:90,2] + -11.139;
   1:L PR[91] 10mm/sec CNT100;
   1:  PR[GP1:91,1] = PR[GP1:90,1] + 58.505;
   1:  PR[GP1:91,2] = PR[GP1:90,2] + -8.396;
   1:L PR[91] 10mm/sec CNT100;
   1:  PR[GP1:91,1] = PR[GP1:90,1] + 59.987;
   1:  PR[GP1:91,2] = PR[GP1:90,2] + 0.296;
   1:L PR[91] 10mm/sec CNT100;
   1:  PR[GP1:91,1] = PR[GP1:90,1] + 59.681;
   1:  PR[GP1:91,2] = PR[GP1:90,2] + 3.008;
   1:L PR[91] 10mm/sec CNT100;
   1:  PR[GP1:91,1] = PR[GP1:90,1] + 58.192;
   1:  PR[GP1:91,2] = PR[GP1:90,2] + 11.699;
   1:L PR[91] 10mm/sec CNT100;
   1:  PR[GP1:91,1] = PR[GP1:90,1] + 57.272;
   1:  PR[GP1:91,2] = PR[GP1:90,2] + 14.201;
   1:L PR[91] 10mm/sec CNT100;
   1:  PR[GP1:91,1] = PR[GP1:90,1] + 52.833;
   1:  PR[GP1:91,2] = PR[GP1:90,2] + 22.204;
   1:L PR[91] 10mm/sec CNT100;
   1:  PR[GP1:91,1] = PR[GP1:90,1] + 51.409;
   1:  PR[GP1:91,2] = PR[GP1:90,2] + 24.414;
   1:L PR[91] 10mm/sec CNT100;
   1:  PR[GP1:91,1] = PR[GP1:90,1] + 49.695;
   1:  PR[GP1:91,2] = PR[GP1:90,2] + 26.092;
   1:L PR[91] 10mm/sec CNT100;
   1:  PR[GP1:91,1] = PR[GP1:90,1] + 42.458;
   1:  PR[GP1:91,2] = PR[GP1:90,2] + 32.642;
   1:L PR[91] 10mm/sec CNT100;
   1:  PR[GP1:91,1] = PR[GP1:90,1] + 40.601;
   1:  PR[GP1:91,2] = PR[GP1:90,2] + 33.807;
   1:L PR[91] 10mm/sec CNT100;
   1:  PR[GP1:91,1] = PR[GP1:90,1] + 30.949;
   1:  PR[GP1:91,2] = PR[GP1:90,2] + 38.024;
   1:L PR[91] 10mm/sec CNT100;
   1:  PR[GP1:91,1] = PR[GP1:90,1] + 29.133;
   1:  PR[GP1:91,2] = PR[GP1:90,2] + 38.687;
   1:L PR[91] 10mm/sec CNT100;
   1:  PR[GP1:91,1] = PR[GP1:90,1] + 27.417;
   1:  PR[GP1:91,2] = PR[GP1:90,2] + 38.930;
   1:L PR[91] 10mm/sec CNT100;
   1:  PR[GP1:91,1] = PR[GP1:90,1] + 16.241;
   1:  PR[GP1:91,2] = PR[GP1:90,2] + 39.968;
   1:L PR[91] 10mm/sec CNT100;
   1:  PR[GP1:91,1] = PR[GP1:90,1] + 14.852;
   1:  PR[GP1:91,2] = PR[GP1:90,2] + 39.876;
   1:L PR[91] 10mm/sec CNT100;
   1:  PR[GP1:91,1] = PR[GP1:90,1] + 3.050;
   1:  PR[GP1:91,2] = PR[GP1:90,2] + 37.089;
   1:L PR[91] 10mm/sec CNT100;
   1:  PR[GP1:91,1] = PR[GP1:90,1] + 2.106;
   1:  PR[GP1:91,2] = PR[GP1:90,2] + 36.817;
   1:L PR[91] 10mm/sec CNT100;
   1:  PR[GP1:91,1] = PR[GP1:90,1] + 0.363;
   1:  PR[GP1:91,2] = PR[GP1:90,2] + 35.900;
   1:L PR[91] 10mm/sec CNT100;
   1:  PR[GP1:91,1] = PR[GP1:90,1] + -0.263;
   1:  PR[GP1:91,2] = PR[GP1:90,2] + 35.391;
   1:L PR[91] 10mm/sec CNT100;
   1:  PR[GP1:91,1] = PR[GP1:90,1] + -0.889;
   1:  PR[GP1:91,2] = PR[GP1:90,2] + 35.900;
   1:L PR[91] 10mm/sec CNT100;
   1:  PR[GP1:91,1] = PR[GP1:90,1] + -2.629;
   1:  PR[GP1:91,2] = PR[GP1:90,2] + 36.818;
   1:L PR[91] 10mm/sec CNT100;
   1:  PR[GP1:91,1] = PR[GP1:90,1] + -3.572;
   1:  PR[GP1:91,2] = PR[GP1:90,2] + 37.089;
   1:L PR[91] 10mm/sec CNT100;
   1:  PR[GP1:91,1] = PR[GP1:90,1] + -15.377;
   1:  PR[GP1:91,2] = PR[GP1:90,2] + 39.876;
   1:L PR[91] 10mm/sec CNT100;
   1:  PR[GP1:91,1] = PR[GP1:90,1] + -16.758;
   1:  PR[GP1:91,2] = PR[GP1:90,2] + 39.967;
   1:L PR[91] 10mm/sec CNT100;
   1:  PR[GP1:91,1] = PR[GP1:90,1] + -18.360;
   1:  PR[GP1:91,2] = PR[GP1:90,2] + 39.745;
   1:L PR[91] 10mm/sec CNT100;
   1:  PR[GP1:91,1] = PR[GP1:90,1] + -29.682;
   1:  PR[GP1:91,2] = PR[GP1:90,2] + 38.681;
   1:L PR[91] 10mm/sec CNT100;
   1:  PR[GP1:91,1] = PR[GP1:90,1] + -31.482;
   1:  PR[GP1:91,2] = PR[GP1:90,2] + 38.021;
   1:L PR[91] 10mm/sec CNT100;
   1:  PR[GP1:91,1] = PR[GP1:90,1] + -41.134;
   1:  PR[GP1:91,2] = PR[GP1:90,2] + 33.801;
   1:L PR[91] 10mm/sec CNT100;
   1:  PR[GP1:91,1] = PR[GP1:90,1] + -42.994;
   1:  PR[GP1:91,2] = PR[GP1:90,2] + 32.629;
   1:L PR[91] 10mm/sec CNT100;
   1:  PR[GP1:91,1] = PR[GP1:90,1] + -44.707;
   1:  PR[GP1:91,2] = PR[GP1:90,2] + 30.957;
   1:L PR[91] 10mm/sec CNT100;
   1:  PR[GP1:91,1] = PR[GP1:90,1] + -51.964;
   1:  PR[GP1:91,2] = PR[GP1:90,2] + 24.386;
   1:L PR[91] 10mm/sec CNT100;
   1:  PR[GP1:91,1] = PR[GP1:90,1] + -53.366;
   1:  PR[GP1:91,2] = PR[GP1:90,2] + 22.197;
   1:L PR[91] 10mm/sec CNT100;
   1:  PR[GP1:91,1] = PR[GP1:90,1] + -57.805;
   1:  PR[GP1:91,2] = PR[GP1:90,2] + 14.179;
   1:L PR[91] 10mm/sec CNT100;
   1:  PR[GP1:91,1] = PR[GP1:90,1] + -58.724;
   1:  PR[GP1:91,2] = PR[GP1:90,2] + 11.648;
   1:L PR[91] 10mm/sec CNT100;
   1:  PR[GP1:91,1] = PR[GP1:90,1] + -59.024;
   1:  PR[GP1:91,2] = PR[GP1:90,2] + 8.963;
   1:L PR[91] 10mm/sec CNT100;
   1:  PR[GP1:91,1] = PR[GP1:90,1] + -60.514;
   1:  PR[GP1:91,2] = PR[GP1:90,2] + 0.261;
   1:L PR[91] 10mm/sec CNT100;
   1:  PR[GP1:91,1] = PR[GP1:90,1] + -60.218;
   1:  PR[GP1:91,2] = PR[GP1:90,2] + -2.391;
   1:L PR[91] 10mm/sec CNT100;
   1:  PR[GP1:91,1] = PR[GP1:90,1] + -58.736;
   1:  PR[GP1:91,2] = PR[GP1:90,2] + -11.056;
   1:L PR[91] 10mm/sec CNT100;
   1:  PR[GP1:91,1] = PR[GP1:90,1] + -57.812;
   1:  PR[GP1:91,2] = PR[GP1:90,2] + -13.603;
   1:L PR[91] 10mm/sec CNT100;
   1:  PR[GP1:91,1] = PR[GP1:90,1] + -53.392;
   1:  PR[GP1:91,2] = PR[GP1:90,2] + -21.606;
   1:L PR[91] 10mm/sec CNT100;
   1:  PR[GP1:91,1] = PR[GP1:90,1] + -51.983;
   1:  PR[GP1:91,2] = PR[GP1:90,2] + -23.806;
   1:L PR[91] 10mm/sec CNT100;
   1:  PR[GP1:91,1] = PR[GP1:90,1] + -50.266;
   1:  PR[GP1:91,2] = PR[GP1:90,2] + -25.490;
   1:L PR[91] 10mm/sec CNT100;
   1:  PR[GP1:91,1] = PR[GP1:90,1] + -43.059;
   1:  PR[GP1:91,2] = PR[GP1:90,2] + -32.029;
   1:L PR[91] 10mm/sec CNT100;
   1:  PR[GP1:91,1] = PR[GP1:90,1] + -41.189;
   1:  PR[GP1:91,2] = PR[GP1:90,2] + -33.208;
   1:L PR[91] 10mm/sec CNT100;
   1:  PR[GP1:91,1] = PR[GP1:90,1] + -31.574;
   1:  PR[GP1:91,2] = PR[GP1:90,2] + -37.439;
   1:L PR[91] 10mm/sec CNT100;
   1:  PR[GP1:91,1] = PR[GP1:90,1] + -29.760;
   1:  PR[GP1:91,2] = PR[GP1:90,2] + -38.104;
   1:L PR[91] 10mm/sec CNT100;
   1:  PR[GP1:91,1] = PR[GP1:90,1] + -28.037;
   1:  PR[GP1:91,2] = PR[GP1:90,2] + -38.349;
   1:L PR[91] 10mm/sec CNT100;
   1:  PR[GP1:91,1] = PR[GP1:90,1] + -16.897;
   1:  PR[GP1:91,2] = PR[GP1:90,2] + -39.418;
   1:L PR[91] 10mm/sec CNT100;
   1:  PR[GP1:91,1] = PR[GP1:90,1] + -15.499;
   1:  PR[GP1:91,2] = PR[GP1:90,2] + -39.325;
   1:L PR[91] 10mm/sec CNT100;
   1:  PR[GP1:91,1] = PR[GP1:90,1] + -3.889;
   1:  PR[GP1:91,2] = PR[GP1:90,2] + -36.669;
   1:L PR[91] 10mm/sec CNT100;
   1:  PR[GP1:91,1] = PR[GP1:90,1] + -2.860;
   1:  PR[GP1:91,2] = PR[GP1:90,2] + -36.374;
   1:L PR[91] 10mm/sec CNT100;
   1:  PR[GP1:91,1] = PR[GP1:90,1] + -0.265;
   1:  PR[GP1:91,2] = PR[GP1:90,2] + -34.853;
   1:L PR[91] 10mm/sec CNT100;
   1:  PR[GP1:91,1] = PR[GP1:90,1] + 2.078;
   1:  PR[GP1:91,2] = PR[GP1:90,2] + -36.443;
   1:  PR[GP1:91,3] = PR[GP1:90,3] + 79.605;
   1:L PR[91] 10mm/sec CNT100;
   1:  PR[GP1:91,1] = PR[GP1:90,1] + 2.987;
   1:  PR[GP1:91,2] = PR[GP1:90,2] + -36.704;
   1:L PR[91] 10mm/sec CNT100;
   1:  PR[GP1:91,1] = PR[GP1:90,1] + 14.797;
   1:  PR[GP1:91,2] = PR[GP1:90,2] + -39.406;
   1:L PR[91] 10mm/sec CNT100;
   1:  PR[GP1:91,1] = PR[GP1:90,1] + 16.054;
   1:  PR[GP1:91,2] = PR[GP1:90,2] + -39.489;
   1:L PR[91] 10mm/sec CNT100;
   1:  PR[GP1:91,1] = PR[GP1:90,1] + 17.516;
   1:  PR[GP1:91,2] = PR[GP1:90,2] + -39.288;
   1:L PR[91] 10mm/sec CNT100;
   1:  PR[GP1:91,1] = PR[GP1:90,1] + 29.020;
   1:  PR[GP1:91,2] = PR[GP1:90,2] + -38.170;
   1:L PR[91] 10mm/sec CNT100;
   1:  PR[GP1:91,1] = PR[GP1:90,1] + 30.696;
   1:  PR[GP1:91,2] = PR[GP1:90,2] + -37.558;
   1:L PR[91] 10mm/sec CNT100;
   1:  PR[GP1:91,1] = PR[GP1:90,1] + 40.510;
   1:  PR[GP1:91,2] = PR[GP1:90,2] + -33.242;
   1:L PR[91] 10mm/sec CNT100;
   1:  PR[GP1:91,1] = PR[GP1:90,1] + 42.248;
   1:  PR[GP1:91,2] = PR[GP1:90,2] + -32.151;
   1:L PR[91] 10mm/sec CNT100;
   1:  PR[GP1:91,1] = PR[GP1:90,1] + 43.858;
   1:  PR[GP1:91,2] = PR[GP1:90,2] + -30.582;
   1:L PR[91] 10mm/sec CNT100;
   1:  PR[GP1:91,1] = PR[GP1:90,1] + 51.253;
   1:  PR[GP1:91,2] = PR[GP1:90,2] + -23.856;
   1:L PR[91] 10mm/sec CNT100;
   1:  PR[GP1:91,1] = PR[GP1:90,1] + 52.597;
   1:  PR[GP1:91,2] = PR[GP1:90,2] + -21.772;
   1:L PR[91] 10mm/sec CNT100;
   1:  PR[GP1:91,1] = PR[GP1:90,1] + 57.124;
   1:  PR[GP1:91,2] = PR[GP1:90,2] + -13.588;
   1:L PR[91] 10mm/sec CNT100;
   1:  PR[GP1:91,1] = PR[GP1:90,1] + 57.993;
   1:  PR[GP1:91,2] = PR[GP1:90,2] + -11.225;
   1:L PR[91] 10mm/sec CNT100;
   1:  PR[GP1:91,1] = PR[GP1:90,1] + 58.290;
   1:  PR[GP1:91,2] = PR[GP1:90,2] + -8.616;
   1:L PR[91] 10mm/sec CNT100;
   1:  PR[GP1:91,1] = PR[GP1:90,1] + 59.810;
   1:  PR[GP1:91,2] = PR[GP1:90,2] + 0.296;
   1:L PR[91] 10mm/sec CNT100;
   1:  PR[GP1:91,1] = PR[GP1:90,1] + 59.518;
   1:  PR[GP1:91,2] = PR[GP1:90,2] + 2.877;
   1:L PR[91] 10mm/sec CNT100;
   1:  PR[GP1:91,1] = PR[GP1:90,1] + 57.993;
   1:  PR[GP1:91,2] = PR[GP1:90,2] + 11.786;
   1:L PR[91] 10mm/sec CNT100;
   1:  PR[GP1:91,1] = PR[GP1:90,1] + 57.118;
   1:  PR[GP1:91,2] = PR[GP1:90,2] + 14.164;
   1:L PR[91] 10mm/sec CNT100;
   1:  PR[GP1:91,1] = PR[GP1:90,1] + 52.571;
   1:  PR[GP1:91,2] = PR[GP1:90,2] + 22.362;
   1:L PR[91] 10mm/sec CNT100;
   1:  PR[GP1:91,1] = PR[GP1:90,1] + 51.221;
   1:  PR[GP1:91,2] = PR[GP1:90,2] + 24.456;
   1:L PR[91] 10mm/sec CNT100;
   1:  PR[GP1:91,1] = PR[GP1:90,1] + 49.597;
   1:  PR[GP1:91,2] = PR[GP1:90,2] + 26.046;
   1:L PR[91] 10mm/sec CNT100;
   1:  PR[GP1:91,1] = PR[GP1:90,1] + 42.201;
   1:  PR[GP1:91,2] = PR[GP1:90,2] + 32.740;
   1:L PR[91] 10mm/sec CNT100;
   1:  PR[GP1:91,1] = PR[GP1:90,1] + 40.454;
   1:  PR[GP1:91,2] = PR[GP1:90,2] + 33.836;
   1:L PR[91] 10mm/sec CNT100;
   1:  PR[GP1:91,1] = PR[GP1:90,1] + 30.603;
   1:  PR[GP1:91,2] = PR[GP1:90,2] + 38.140;
   1:L PR[91] 10mm/sec CNT100;
   1:  PR[GP1:91,1] = PR[GP1:90,1] + 28.914;
   1:  PR[GP1:91,2] = PR[GP1:90,2] + 38.757;
   1:L PR[91] 10mm/sec CNT100;
   1:  PR[GP1:91,1] = PR[GP1:90,1] + 27.318;
   1:  PR[GP1:91,2] = PR[GP1:90,2] + 38.983;
   1:L PR[91] 10mm/sec CNT100;
   1:  PR[GP1:91,1] = PR[GP1:90,1] + 15.939;
   1:  PR[GP1:91,2] = PR[GP1:90,2] + 40.040;
   1:L PR[91] 10mm/sec CNT100;
   1:  PR[GP1:91,1] = PR[GP1:90,1] + 14.673;
   1:  PR[GP1:91,2] = PR[GP1:90,2] + 39.956;
   1:L PR[91] 10mm/sec CNT100;
   1:  PR[GP1:91,1] = PR[GP1:90,1] + 2.670;
   1:  PR[GP1:91,2] = PR[GP1:90,2] + 37.121;
   1:L PR[91] 10mm/sec CNT100;
   1:  PR[GP1:91,1] = PR[GP1:90,1] + 1.847;
   1:  PR[GP1:91,2] = PR[GP1:90,2] + 36.885;
   1:L PR[91] 10mm/sec CNT100;
   1:  PR[GP1:91,1] = PR[GP1:90,1] + 0.190;
   1:  PR[GP1:91,2] = PR[GP1:90,2] + 36.014;
   1:L PR[91] 10mm/sec CNT100;
   1:  PR[GP1:91,1] = PR[GP1:90,1] + -0.263;
   1:  PR[GP1:91,2] = PR[GP1:90,2] + 35.646;
   1:L PR[91] 10mm/sec CNT100;
   1:  PR[GP1:91,1] = PR[GP1:90,1] + -0.716;
   1:  PR[GP1:91,2] = PR[GP1:90,2] + 36.014;
   1:L PR[91] 10mm/sec CNT100;
   1:  PR[GP1:91,1] = PR[GP1:90,1] + -2.371;
   1:  PR[GP1:91,2] = PR[GP1:90,2] + 36.885;
   1:L PR[91] 10mm/sec CNT100;
   1:  PR[GP1:91,1] = PR[GP1:90,1] + -3.191;
   1:  PR[GP1:91,2] = PR[GP1:90,2] + 37.121;
   1:L PR[91] 10mm/sec CNT100;
   1:  PR[GP1:91,1] = PR[GP1:90,1] + -15.198;
   1:  PR[GP1:91,2] = PR[GP1:90,2] + 39.956;
   1:L PR[91] 10mm/sec CNT100;
   1:  PR[GP1:91,1] = PR[GP1:90,1] + -16.455;
   1:  PR[GP1:91,2] = PR[GP1:90,2] + 40.039;
   1:L PR[91] 10mm/sec CNT100;
   1:  PR[GP1:91,1] = PR[GP1:90,1] + -17.920;
   1:  PR[GP1:91,2] = PR[GP1:90,2] + 39.836;
   1:L PR[91] 10mm/sec CNT100;
   1:  PR[GP1:91,1] = PR[GP1:90,1] + -29.462;
   1:  PR[GP1:91,2] = PR[GP1:90,2] + 38.751;
   1:L PR[91] 10mm/sec CNT100;
   1:  PR[GP1:91,1] = PR[GP1:90,1] + -31.136;
   1:  PR[GP1:91,2] = PR[GP1:90,2] + 38.138;
   1:L PR[91] 10mm/sec CNT100;
   1:  PR[GP1:91,1] = PR[GP1:90,1] + -40.987;
   1:  PR[GP1:91,2] = PR[GP1:90,2] + 33.831;
   1:L PR[91] 10mm/sec CNT100;
   1:  PR[GP1:91,1] = PR[GP1:90,1] + -42.736;
   1:  PR[GP1:91,2] = PR[GP1:90,2] + 32.728;
   1:L PR[91] 10mm/sec CNT100;
   1:  PR[GP1:91,1] = PR[GP1:90,1] + -44.349;
   1:  PR[GP1:91,2] = PR[GP1:90,2] + 31.153;
   1:L PR[91] 10mm/sec CNT100;
   1:  PR[GP1:91,1] = PR[GP1:90,1] + -51.775;
   1:  PR[GP1:91,2] = PR[GP1:90,2] + 24.430;
   1:L PR[91] 10mm/sec CNT100;
   1:  PR[GP1:91,1] = PR[GP1:90,1] + -53.104;
   1:  PR[GP1:91,2] = PR[GP1:90,2] + 22.356;
   1:L PR[91] 10mm/sec CNT100;
   1:  PR[GP1:91,1] = PR[GP1:90,1] + -57.651;
   1:  PR[GP1:91,2] = PR[GP1:90,2] + 14.143;
   1:L PR[91] 10mm/sec CNT100;
   1:  PR[GP1:91,1] = PR[GP1:90,1] + -58.523;
   1:  PR[GP1:91,2] = PR[GP1:90,2] + 11.738;
   1:L PR[91] 10mm/sec CNT100;
   1:  PR[GP1:91,1] = PR[GP1:90,1] + -58.810;
   1:  PR[GP1:91,2] = PR[GP1:90,2] + 9.183;
   1:L PR[91] 10mm/sec CNT100;
   1:  PR[GP1:91,1] = PR[GP1:90,1] + -60.336;
   1:  PR[GP1:91,2] = PR[GP1:90,2] + 0.261;
   1:L PR[91] 10mm/sec CNT100;
   1:  PR[GP1:91,1] = PR[GP1:90,1] + -60.055;
   1:  PR[GP1:91,2] = PR[GP1:90,2] + -2.263;
   1:L PR[91] 10mm/sec CNT100;
   1:  PR[GP1:91,1] = PR[GP1:90,1] + -58.536;
   1:  PR[GP1:91,2] = PR[GP1:90,2] + -11.145;
   1:L PR[91] 10mm/sec CNT100;
   1:  PR[GP1:91,1] = PR[GP1:90,1] + -57.657;
   1:  PR[GP1:91,2] = PR[GP1:90,2] + -13.566;
   1:L PR[91] 10mm/sec CNT100;
   1:  PR[GP1:91,1] = PR[GP1:90,1] + -53.130;
   1:  PR[GP1:91,2] = PR[GP1:90,2] + -21.765;
   1:L PR[91] 10mm/sec CNT100;
   1:  PR[GP1:91,1] = PR[GP1:90,1] + -51.795;
   1:  PR[GP1:91,2] = PR[GP1:90,2] + -23.849;
   1:L PR[91] 10mm/sec CNT100;
   1:  PR[GP1:91,1] = PR[GP1:90,1] + -50.168;
   1:  PR[GP1:91,2] = PR[GP1:90,2] + -25.445;
   1:L PR[91] 10mm/sec CNT100;
   1:  PR[GP1:91,1] = PR[GP1:90,1] + -42.802;
   1:  PR[GP1:91,2] = PR[GP1:90,2] + -32.127;
   1:L PR[91] 10mm/sec CNT100;
   1:  PR[GP1:91,1] = PR[GP1:90,1] + -41.043;
   1:  PR[GP1:91,2] = PR[GP1:90,2] + -33.236;
   1:L PR[91] 10mm/sec CNT100;
   1:  PR[GP1:91,1] = PR[GP1:90,1] + -31.229;
   1:  PR[GP1:91,2] = PR[GP1:90,2] + -37.555;
   1:L PR[91] 10mm/sec CNT100;
   1:  PR[GP1:91,1] = PR[GP1:90,1] + -29.542;
   1:  PR[GP1:91,2] = PR[GP1:90,2] + -38.173;
   1:L PR[91] 10mm/sec CNT100;
   1:  PR[GP1:91,1] = PR[GP1:90,1] + -27.940;
   1:  PR[GP1:91,2] = PR[GP1:90,2] + -38.401;
   1:L PR[91] 10mm/sec CNT100;
   1:  PR[GP1:91,1] = PR[GP1:90,1] + -16.596;
   1:  PR[GP1:91,2] = PR[GP1:90,2] + -39.490;
   1:L PR[91] 10mm/sec CNT100;
   1:  PR[GP1:91,1] = PR[GP1:90,1] + -15.323;
   1:  PR[GP1:91,2] = PR[GP1:90,2] + -39.406;
   1:L PR[91] 10mm/sec CNT100;
   1:  PR[GP1:91,1] = PR[GP1:90,1] + -3.513;
   1:  PR[GP1:91,2] = PR[GP1:90,2] + -36.704;
   1:L PR[91] 10mm/sec CNT100;
   1:  PR[GP1:91,1] = PR[GP1:90,1] + -2.606;
   1:  PR[GP1:91,2] = PR[GP1:90,2] + -36.443;
   1:L PR[91] 10mm/sec CNT100;
   1:  PR[GP1:91,1] = PR[GP1:90,1] + -0.264;
   1:  PR[GP1:91,2] = PR[GP1:90,2] + -35.071;
   1:L PR[91] 10mm/sec CNT100;
   1:  PR[GP1:91,1] = PR[GP1:90,1] + 1.823;
   1:  PR[GP1:91,2] = PR[GP1:90,2] + -36.512;
   1:  PR[GP1:91,3] = PR[GP1:90,3] + 80.215;
   1:L PR[91] 10mm/sec CNT100;
   1:  PR[GP1:91,1] = PR[GP1:90,1] + 2.612;
   1:  PR[GP1:91,2] = PR[GP1:90,2] + -36.738;
   1:L PR[91] 10mm/sec CNT100;
   1:  PR[GP1:91,1] = PR[GP1:90,1] + 14.620;
   1:  PR[GP1:91,2] = PR[GP1:90,2] + -39.486;
   1:L PR[91] 10mm/sec CNT100;
   1:  PR[GP1:91,1] = PR[GP1:90,1] + 15.754;
   1:  PR[GP1:91,2] = PR[GP1:90,2] + -39.561;
   1:L PR[91] 10mm/sec CNT100;
   1:  PR[GP1:91,1] = PR[GP1:90,1] + 17.080;
   1:  PR[GP1:91,2] = PR[GP1:90,2] + -39.378;
   1:L PR[91] 10mm/sec CNT100;
   1:  PR[GP1:91,1] = PR[GP1:90,1] + 28.802;
   1:  PR[GP1:91,2] = PR[GP1:90,2] + -38.239;
   1:L PR[91] 10mm/sec CNT100;
   1:  PR[GP1:91,1] = PR[GP1:90,1] + 30.352;
   1:  PR[GP1:91,2] = PR[GP1:90,2] + -37.673;
   1:L PR[91] 10mm/sec CNT100;
   1:  PR[GP1:91,1] = PR[GP1:90,1] + 40.365;
   1:  PR[GP1:91,2] = PR[GP1:90,2] + -33.270;
   1:L PR[91] 10mm/sec CNT100;
   1:  PR[GP1:91,1] = PR[GP1:90,1] + 41.993;
   1:  PR[GP1:91,2] = PR[GP1:90,2] + -32.249;
   1:L PR[91] 10mm/sec CNT100;
   1:  PR[GP1:91,1] = PR[GP1:90,1] + 43.503;
   1:  PR[GP1:91,2] = PR[GP1:90,2] + -30.777;
   1:L PR[91] 10mm/sec CNT100;
   1:  PR[GP1:91,1] = PR[GP1:90,1] + 51.066;
   1:  PR[GP1:91,2] = PR[GP1:90,2] + -23.897;
   1:L PR[91] 10mm/sec CNT100;
   1:  PR[GP1:91,1] = PR[GP1:90,1] + 52.335;
   1:  PR[GP1:91,2] = PR[GP1:90,2] + -21.929;
   1:L PR[91] 10mm/sec CNT100;
   1:  PR[GP1:91,1] = PR[GP1:90,1] + 56.970;
   1:  PR[GP1:91,2] = PR[GP1:90,2] + -13.551;
   1:L PR[91] 10mm/sec CNT100;
   1:  PR[GP1:91,1] = PR[GP1:90,1] + 57.794;
   1:  PR[GP1:91,2] = PR[GP1:90,2] + -11.312;
   1:L PR[91] 10mm/sec CNT100;
   1:  PR[GP1:91,1] = PR[GP1:90,1] + 58.075;
   1:  PR[GP1:91,2] = PR[GP1:90,2] + -8.836;
   1:L PR[91] 10mm/sec CNT100;
   1:  PR[GP1:91,1] = PR[GP1:90,1] + 59.633;
   1:  PR[GP1:91,2] = PR[GP1:90,2] + 0.296;
   1:L PR[91] 10mm/sec CNT100;
   1:  PR[GP1:91,1] = PR[GP1:90,1] + 59.356;
   1:  PR[GP1:91,2] = PR[GP1:90,2] + 2.746;
   1:L PR[91] 10mm/sec CNT100;
   1:  PR[GP1:91,1] = PR[GP1:90,1] + 57.793;
   1:  PR[GP1:91,2] = PR[GP1:90,2] + 11.873;
   1:L PR[91] 10mm/sec CNT100;
   1:  PR[GP1:91,1] = PR[GP1:90,1] + 56.964;
   1:  PR[GP1:91,2] = PR[GP1:90,2] + 14.128;
   1:L PR[91] 10mm/sec CNT100;
   1:  PR[GP1:91,1] = PR[GP1:90,1] + 52.309;
   1:  PR[GP1:91,2] = PR[GP1:90,2] + 22.521;
   1:L PR[91] 10mm/sec CNT100;
   1:  PR[GP1:91,1] = PR[GP1:90,1] + 51.034;
   1:  PR[GP1:91,2] = PR[GP1:90,2] + 24.498;
   1:L PR[91] 10mm/sec CNT100;
   1:  PR[GP1:91,1] = PR[GP1:90,1] + 49.500;
   1:  PR[GP1:91,2] = PR[GP1:90,2] + 26.000;
   1:L PR[91] 10mm/sec CNT100;
   1:  PR[GP1:91,1] = PR[GP1:90,1] + 41.945;
   1:  PR[GP1:91,2] = PR[GP1:90,2] + 32.838;
   1:L PR[91] 10mm/sec CNT100;
   1:  PR[GP1:91,1] = PR[GP1:90,1] + 40.308;
   1:  PR[GP1:91,2] = PR[GP1:90,2] + 33.865;
   1:L PR[91] 10mm/sec CNT100;
   1:  PR[GP1:91,1] = PR[GP1:90,1] + 30.257;
   1:  PR[GP1:91,2] = PR[GP1:90,2] + 38.257;
   1:L PR[91] 10mm/sec CNT100;
   1:  PR[GP1:91,1] = PR[GP1:90,1] + 28.695;
   1:  PR[GP1:91,2] = PR[GP1:90,2] + 38.827;
   1:L PR[91] 10mm/sec CNT100;
   1:  PR[GP1:91,1] = PR[GP1:90,1] + 27.219;
   1:  PR[GP1:91,2] = PR[GP1:90,2] + 39.036;
   1:L PR[91] 10mm/sec CNT100;
   1:  PR[GP1:91,1] = PR[GP1:90,1] + 15.637;
   1:  PR[GP1:91,2] = PR[GP1:90,2] + 40.112;
   1:L PR[91] 10mm/sec CNT100;
   1:  PR[GP1:91,1] = PR[GP1:90,1] + 14.494;
   1:  PR[GP1:91,2] = PR[GP1:90,2] + 40.036;
   1:L PR[91] 10mm/sec CNT100;
   1:  PR[GP1:91,1] = PR[GP1:90,1] + 2.289;
   1:  PR[GP1:91,2] = PR[GP1:90,2] + 37.154;
   1:L PR[91] 10mm/sec CNT100;
   1:  PR[GP1:91,1] = PR[GP1:90,1] + 1.589;
   1:  PR[GP1:91,2] = PR[GP1:90,2] + 36.952;
   1:L PR[91] 10mm/sec CNT100;
   1:  PR[GP1:91,1] = PR[GP1:90,1] + -0.264;
   1:  PR[GP1:91,2] = PR[GP1:90,2] + 35.981;
   1:L PR[91] 10mm/sec CNT100;
   1:  PR[GP1:91,1] = PR[GP1:90,1] + -2.112;
   1:  PR[GP1:91,2] = PR[GP1:90,2] + 36.953;
   1:L PR[91] 10mm/sec CNT100;
   1:  PR[GP1:91,1] = PR[GP1:90,1] + -2.811;
   1:  PR[GP1:91,2] = PR[GP1:90,2] + 37.154;
   1:L PR[91] 10mm/sec CNT100;
   1:  PR[GP1:91,1] = PR[GP1:90,1] + -15.019;
   1:  PR[GP1:91,2] = PR[GP1:90,2] + 40.036;
   1:L PR[91] 10mm/sec CNT100;
   1:  PR[GP1:91,1] = PR[GP1:90,1] + -16.152;
   1:  PR[GP1:91,2] = PR[GP1:90,2] + 40.111;
   1:L PR[91] 10mm/sec CNT100;
   1:  PR[GP1:91,1] = PR[GP1:90,1] + -17.481;
   1:  PR[GP1:91,2] = PR[GP1:90,2] + 39.927;
   1:L PR[91] 10mm/sec CNT100;
   1:  PR[GP1:91,1] = PR[GP1:90,1] + -29.242;
   1:  PR[GP1:91,2] = PR[GP1:90,2] + 38.821;
   1:L PR[91] 10mm/sec CNT100;
   1:  PR[GP1:91,1] = PR[GP1:90,1] + -30.789;
   1:  PR[GP1:91,2] = PR[GP1:90,2] + 38.255;
   1:L PR[91] 10mm/sec CNT100;
   1:  PR[GP1:91,1] = PR[GP1:90,1] + -40.841;
   1:  PR[GP1:91,2] = PR[GP1:90,2] + 33.860;
   1:L PR[91] 10mm/sec CNT100;
   1:  PR[GP1:91,1] = PR[GP1:90,1] + -42.478;
   1:  PR[GP1:91,2] = PR[GP1:90,2] + 32.827;
   1:L PR[91] 10mm/sec CNT100;
   1:  PR[GP1:91,1] = PR[GP1:90,1] + -43.991;
   1:  PR[GP1:91,2] = PR[GP1:90,2] + 31.350;
   1:L PR[91] 10mm/sec CNT100;
   1:  PR[GP1:91,1] = PR[GP1:90,1] + -51.586;
   1:  PR[GP1:91,2] = PR[GP1:90,2] + 24.473;
   1:L PR[91] 10mm/sec CNT100;
   1:  PR[GP1:91,1] = PR[GP1:90,1] + -52.841;
   1:  PR[GP1:91,2] = PR[GP1:90,2] + 22.515;
   1:L PR[91] 10mm/sec CNT100;
   1:  PR[GP1:91,1] = PR[GP1:90,1] + -57.496;
   1:  PR[GP1:91,2] = PR[GP1:90,2] + 14.107;
   1:L PR[91] 10mm/sec CNT100;
   1:  PR[GP1:91,1] = PR[GP1:90,1] + -58.323;
   1:  PR[GP1:91,2] = PR[GP1:90,2] + 11.828;
   1:L PR[91] 10mm/sec CNT100;
   1:  PR[GP1:91,1] = PR[GP1:90,1] + -58.595;
   1:  PR[GP1:91,2] = PR[GP1:90,2] + 9.403;
   1:L PR[91] 10mm/sec CNT100;
   1:  PR[GP1:91,1] = PR[GP1:90,1] + -60.159;
   1:  PR[GP1:91,2] = PR[GP1:90,2] + 0.261;
   1:L PR[91] 10mm/sec CNT100;
   1:  PR[GP1:91,1] = PR[GP1:90,1] + -59.892;
   1:  PR[GP1:91,2] = PR[GP1:90,2] + -2.135;
   1:L PR[91] 10mm/sec CNT100;
   1:  PR[GP1:91,1] = PR[GP1:90,1] + -58.336;
   1:  PR[GP1:91,2] = PR[GP1:90,2] + -11.234;
   1:L PR[91] 10mm/sec CNT100;
   1:  PR[GP1:91,1] = PR[GP1:90,1] + -57.503;
   1:  PR[GP1:91,2] = PR[GP1:90,2] + -13.530;
   1:L PR[91] 10mm/sec CNT100;
   1:  PR[GP1:91,1] = PR[GP1:90,1] + -52.868;
   1:  PR[GP1:91,2] = PR[GP1:90,2] + -21.923;
   1:L PR[91] 10mm/sec CNT100;
   1:  PR[GP1:91,1] = PR[GP1:90,1] + -51.606;
   1:  PR[GP1:91,2] = PR[GP1:90,2] + -23.892;
   1:L PR[91] 10mm/sec CNT100;
   1:  PR[GP1:91,1] = PR[GP1:90,1] + -50.070;
   1:  PR[GP1:91,2] = PR[GP1:90,2] + -25.399;
   1:L PR[91] 10mm/sec CNT100;
   1:  PR[GP1:91,1] = PR[GP1:90,1] + -42.545;
   1:  PR[GP1:91,2] = PR[GP1:90,2] + -32.226;
   1:L PR[91] 10mm/sec CNT100;
   1:  PR[GP1:91,1] = PR[GP1:90,1] + -40.898;
   1:  PR[GP1:91,2] = PR[GP1:90,2] + -33.265;
   1:L PR[91] 10mm/sec CNT100;
   1:  PR[GP1:91,1] = PR[GP1:90,1] + -30.885;
   1:  PR[GP1:91,2] = PR[GP1:90,2] + -37.671;
   1:L PR[91] 10mm/sec CNT100;
   1:  PR[GP1:91,1] = PR[GP1:90,1] + -29.324;
   1:  PR[GP1:91,2] = PR[GP1:90,2] + -38.243;
   1:L PR[91] 10mm/sec CNT100;
   1:  PR[GP1:91,1] = PR[GP1:90,1] + -27.842;
   1:  PR[GP1:91,2] = PR[GP1:90,2] + -38.454;
   1:L PR[91] 10mm/sec CNT100;
   1:  PR[GP1:91,1] = PR[GP1:90,1] + -16.296;
   1:  PR[GP1:91,2] = PR[GP1:90,2] + -39.562;
   1:L PR[91] 10mm/sec CNT100;
   1:  PR[GP1:91,1] = PR[GP1:90,1] + -15.146;
   1:  PR[GP1:91,2] = PR[GP1:90,2] + -39.486;
   1:L PR[91] 10mm/sec CNT100;
   1:  PR[GP1:91,1] = PR[GP1:90,1] + -3.138;
   1:  PR[GP1:91,2] = PR[GP1:90,2] + -36.738;
   1:L PR[91] 10mm/sec CNT100;
   1:  PR[GP1:91,1] = PR[GP1:90,1] + -2.351;
   1:  PR[GP1:91,2] = PR[GP1:90,2] + -36.512;
   1:L PR[91] 10mm/sec CNT100;
   1:  PR[GP1:91,1] = PR[GP1:90,1] + -0.264;
   1:  PR[GP1:91,2] = PR[GP1:90,2] + -35.290;
   1:L PR[91] 10mm/sec CNT100;
   1:  PR[GP1:91,1] = PR[GP1:90,1] + 1.569;
   1:  PR[GP1:91,2] = PR[GP1:90,2] + -36.581;
   1:  PR[GP1:91,3] = PR[GP1:90,3] + 80.825;
   1:L PR[91] 10mm/sec CNT100;
   1:  PR[GP1:91,1] = PR[GP1:90,1] + 2.236;
   1:  PR[GP1:91,2] = PR[GP1:90,2] + -36.773;
   1:L PR[91] 10mm/sec CNT100;
   1:  PR[GP1:91,1] = PR[GP1:90,1] + 14.443;
   1:  PR[GP1:91,2] = PR[GP1:90,2] + -39.566;
   1:L PR[91] 10mm/sec CNT100;
   1:  PR[GP1:91,1] = PR[GP1:90,1] + 15.454;
   1:  PR[GP1:91,2] = PR[GP1:90,2] + -39.633;
   1:L PR[91] 10mm/sec CNT100;
   1:  PR[GP1:91,1] = PR[GP1:90,1] + 16.643;
   1:  PR[GP1:91,2] = PR[GP1:90,2] + -39.469;
   1:L PR[91] 10mm/sec CNT100;
   1:  PR[GP1:91,1] = PR[GP1:90,1] + 28.585;
   1:  PR[GP1:91,2] = PR[GP1:90,2] + -38.309;
   1:L PR[91] 10mm/sec CNT100;
   1:  PR[GP1:91,1] = PR[GP1:90,1] + 30.008;
   1:  PR[GP1:91,2] = PR[GP1:90,2] + -37.789;
   1:L PR[91] 10mm/sec CNT100;
   1:  PR[GP1:91,1] = PR[GP1:90,1] + 40.220;
   1:  PR[GP1:91,2] = PR[GP1:90,2] + -33.298;
   1:L PR[91] 10mm/sec CNT100;
   1:  PR[GP1:91,1] = PR[GP1:90,1] + 41.737;
   1:  PR[GP1:91,2] = PR[GP1:90,2] + -32.346;
   1:L PR[91] 10mm/sec CNT100;
   1:  PR[GP1:91,1] = PR[GP1:90,1] + 43.148;
   1:  PR[GP1:91,2] = PR[GP1:90,2] + -30.971;
   1:L PR[91] 10mm/sec CNT100;
   1:  PR[GP1:91,1] = PR[GP1:90,1] + 50.879;
   1:  PR[GP1:91,2] = PR[GP1:90,2] + -23.939;
   1:L PR[91] 10mm/sec CNT100;
   1:  PR[GP1:91,1] = PR[GP1:90,1] + 52.073;
   1:  PR[GP1:91,2] = PR[GP1:90,2] + -22.087;
   1:L PR[91] 10mm/sec CNT100;
   1:  PR[GP1:91,1] = PR[GP1:90,1] + 56.816;
   1:  PR[GP1:91,2] = PR[GP1:90,2] + -13.514;
   1:L PR[91] 10mm/sec CNT100;
   1:  PR[GP1:91,1] = PR[GP1:90,1] + 57.594;
   1:  PR[GP1:91,2] = PR[GP1:90,2] + -11.399;
   1:L PR[91] 10mm/sec CNT100;
   1:  PR[GP1:91,1] = PR[GP1:90,1] + 57.860;
   1:  PR[GP1:91,2] = PR[GP1:90,2] + -9.055;
   1:L PR[91] 10mm/sec CNT100;
   1:  PR[GP1:91,1] = PR[GP1:90,1] + 59.455;
   1:  PR[GP1:91,2] = PR[GP1:90,2] + 0.296;
   1:L PR[91] 10mm/sec CNT100;
   1:  PR[GP1:91,1] = PR[GP1:90,1] + 59.193;
   1:  PR[GP1:91,2] = PR[GP1:90,2] + 2.616;
   1:L PR[91] 10mm/sec CNT100;
   1:  PR[GP1:91,1] = PR[GP1:90,1] + 57.593;
   1:  PR[GP1:91,2] = PR[GP1:90,2] + 11.960;
   1:L PR[91] 10mm/sec CNT100;
   1:  PR[GP1:91,1] = PR[GP1:90,1] + 56.809;
   1:  PR[GP1:91,2] = PR[GP1:90,2] + 14.091;
   1:L PR[91] 10mm/sec CNT100;
   1:  PR[GP1:91,1] = PR[GP1:90,1] + 52.046;
   1:  PR[GP1:91,2] = PR[GP1:90,2] + 22.679;
   1:L PR[91] 10mm/sec CNT100;
   1:  PR[GP1:91,1] = PR[GP1:90,1] + 50.846;
   1:  PR[GP1:91,2] = PR[GP1:90,2] + 24.541;
   1:L PR[91] 10mm/sec CNT100;
   1:  PR[GP1:91,1] = PR[GP1:90,1] + 49.403;
   1:  PR[GP1:91,2] = PR[GP1:90,2] + 25.954;
   1:L PR[91] 10mm/sec CNT100;
   1:  PR[GP1:91,1] = PR[GP1:90,1] + 41.688;
   1:  PR[GP1:91,2] = PR[GP1:90,2] + 32.937;
   1:L PR[91] 10mm/sec CNT100;
   1:  PR[GP1:91,1] = PR[GP1:90,1] + 40.162;
   1:  PR[GP1:91,2] = PR[GP1:90,2] + 33.894;
   1:L PR[91] 10mm/sec CNT100;
   1:  PR[GP1:91,1] = PR[GP1:90,1] + 29.911;
   1:  PR[GP1:91,2] = PR[GP1:90,2] + 38.373;
   1:L PR[91] 10mm/sec CNT100;
   1:  PR[GP1:91,1] = PR[GP1:90,1] + 28.476;
   1:  PR[GP1:91,2] = PR[GP1:90,2] + 38.897;
   1:L PR[91] 10mm/sec CNT100;
   1:  PR[GP1:91,1] = PR[GP1:90,1] + 27.120;
   1:  PR[GP1:91,2] = PR[GP1:90,2] + 39.089;
   1:L PR[91] 10mm/sec CNT100;
   1:  PR[GP1:91,1] = PR[GP1:90,1] + 15.335;
   1:  PR[GP1:91,2] = PR[GP1:90,2] + 40.184;
   1:L PR[91] 10mm/sec CNT100;
   1:  PR[GP1:91,1] = PR[GP1:90,1] + 14.315;
   1:  PR[GP1:91,2] = PR[GP1:90,2] + 40.116;
   1:L PR[91] 10mm/sec CNT100;
   1:  PR[GP1:91,1] = PR[GP1:90,1] + 1.908;
   1:  PR[GP1:91,2] = PR[GP1:90,2] + 37.186;
   1:L PR[91] 10mm/sec CNT100;
   1:  PR[GP1:91,1] = PR[GP1:90,1] + 1.331;
   1:  PR[GP1:91,2] = PR[GP1:90,2] + 37.020;
   1:L PR[91] 10mm/sec CNT100;
   1:  PR[GP1:91,1] = PR[GP1:90,1] + -0.263;
   1:  PR[GP1:91,2] = PR[GP1:90,2] + 36.184;
   1:L PR[91] 10mm/sec CNT100;
   1:  PR[GP1:91,1] = PR[GP1:90,1] + -1.854;
   1:  PR[GP1:91,2] = PR[GP1:90,2] + 37.020;
   1:L PR[91] 10mm/sec CNT100;
   1:  PR[GP1:91,1] = PR[GP1:90,1] + -2.430;
   1:  PR[GP1:91,2] = PR[GP1:90,2] + 37.186;
   1:L PR[91] 10mm/sec CNT100;
   1:  PR[GP1:91,1] = PR[GP1:90,1] + -14.840;
   1:  PR[GP1:91,2] = PR[GP1:90,2] + 40.116;
   1:L PR[91] 10mm/sec CNT100;
   1:  PR[GP1:91,1] = PR[GP1:90,1] + -15.850;
   1:  PR[GP1:91,2] = PR[GP1:90,2] + 40.182;
   1:L PR[91] 10mm/sec CNT100;
   1:  PR[GP1:91,1] = PR[GP1:90,1] + -17.041;
   1:  PR[GP1:91,2] = PR[GP1:90,2] + 40.017;
   1:L PR[91] 10mm/sec CNT100;
   1:  PR[GP1:91,1] = PR[GP1:90,1] + -29.023;
   1:  PR[GP1:91,2] = PR[GP1:90,2] + 38.891;
   1:L PR[91] 10mm/sec CNT100;
   1:  PR[GP1:91,1] = PR[GP1:90,1] + -30.443;
   1:  PR[GP1:91,2] = PR[GP1:90,2] + 38.371;
   1:L PR[91] 10mm/sec CNT100;
   1:  PR[GP1:91,1] = PR[GP1:90,1] + -40.694;
   1:  PR[GP1:91,2] = PR[GP1:90,2] + 33.889;
   1:L PR[91] 10mm/sec CNT100;
   1:  PR[GP1:91,1] = PR[GP1:90,1] + -42.220;
   1:  PR[GP1:91,2] = PR[GP1:90,2] + 32.927;
   1:L PR[91] 10mm/sec CNT100;
   1:  PR[GP1:91,1] = PR[GP1:90,1] + -43.634;
   1:  PR[GP1:91,2] = PR[GP1:90,2] + 31.546;
   1:L PR[91] 10mm/sec CNT100;
   1:  PR[GP1:91,1] = PR[GP1:90,1] + -51.398;
   1:  PR[GP1:91,2] = PR[GP1:90,2] + 24.517;
   1:L PR[91] 10mm/sec CNT100;
   1:  PR[GP1:91,1] = PR[GP1:90,1] + -52.578;
   1:  PR[GP1:91,2] = PR[GP1:90,2] + 22.674;
   1:L PR[91] 10mm/sec CNT100;
   1:  PR[GP1:91,1] = PR[GP1:90,1] + -57.341;
   1:  PR[GP1:91,2] = PR[GP1:90,2] + 14.071;
   1:L PR[91] 10mm/sec CNT100;
   1:  PR[GP1:91,1] = PR[GP1:90,1] + -58.123;
   1:  PR[GP1:91,2] = PR[GP1:90,2] + 11.918;
   1:L PR[91] 10mm/sec CNT100;
   1:  PR[GP1:91,1] = PR[GP1:90,1] + -58.380;
   1:  PR[GP1:91,2] = PR[GP1:90,2] + 9.623;
   1:L PR[91] 10mm/sec CNT100;
   1:  PR[GP1:91,1] = PR[GP1:90,1] + -59.982;
   1:  PR[GP1:91,2] = PR[GP1:90,2] + 0.261;
   1:L PR[91] 10mm/sec CNT100;
   1:  PR[GP1:91,1] = PR[GP1:90,1] + -59.729;
   1:  PR[GP1:91,2] = PR[GP1:90,2] + -2.007;
   1:L PR[91] 10mm/sec CNT100;
   1:  PR[GP1:91,1] = PR[GP1:90,1] + -58.136;
   1:  PR[GP1:91,2] = PR[GP1:90,2] + -11.323;
   1:L PR[91] 10mm/sec CNT100;
   1:  PR[GP1:91,1] = PR[GP1:90,1] + -57.348;
   1:  PR[GP1:91,2] = PR[GP1:90,2] + -13.494;
   1:L PR[91] 10mm/sec CNT100;
   1:  PR[GP1:91,1] = PR[GP1:90,1] + -52.606;
   1:  PR[GP1:91,2] = PR[GP1:90,2] + -22.082;
   1:L PR[91] 10mm/sec CNT100;
   1:  PR[GP1:91,1] = PR[GP1:90,1] + -51.418;
   1:  PR[GP1:91,2] = PR[GP1:90,2] + -23.935;
   1:L PR[91] 10mm/sec CNT100;
   1:  PR[GP1:91,1] = PR[GP1:90,1] + -49.972;
   1:  PR[GP1:91,2] = PR[GP1:90,2] + -25.353;
   1:L PR[91] 10mm/sec CNT100;
   1:  PR[GP1:91,1] = PR[GP1:90,1] + -42.288;
   1:  PR[GP1:91,2] = PR[GP1:90,2] + -32.324;
   1:L PR[91] 10mm/sec CNT100;
   1:  PR[GP1:91,1] = PR[GP1:90,1] + -40.752;
   1:  PR[GP1:91,2] = PR[GP1:90,2] + -33.293;
   1:L PR[91] 10mm/sec CNT100;
   1:  PR[GP1:91,1] = PR[GP1:90,1] + -30.540;
   1:  PR[GP1:91,2] = PR[GP1:90,2] + -37.787;
   1:L PR[91] 10mm/sec CNT100;
   1:  PR[GP1:91,1] = PR[GP1:90,1] + -29.106;
   1:  PR[GP1:91,2] = PR[GP1:90,2] + -38.313;
   1:L PR[91] 10mm/sec CNT100;
   1:  PR[GP1:91,1] = PR[GP1:90,1] + -27.744;
   1:  PR[GP1:91,2] = PR[GP1:90,2] + -38.507;
   1:L PR[91] 10mm/sec CNT100;
   1:  PR[GP1:91,1] = PR[GP1:90,1] + -15.996;
   1:  PR[GP1:91,2] = PR[GP1:90,2] + -39.634;
   1:L PR[91] 10mm/sec CNT100;
   1:  PR[GP1:91,1] = PR[GP1:90,1] + -14.969;
   1:  PR[GP1:91,2] = PR[GP1:90,2] + -39.566;
   1:L PR[91] 10mm/sec CNT100;
   1:  PR[GP1:91,1] = PR[GP1:90,1] + -2.763;
   1:  PR[GP1:91,2] = PR[GP1:90,2] + -36.773;
   1:L PR[91] 10mm/sec CNT100;
   1:  PR[GP1:91,1] = PR[GP1:90,1] + -2.096;
   1:  PR[GP1:91,2] = PR[GP1:90,2] + -36.582;
   1:L PR[91] 10mm/sec CNT100;
   1:  PR[GP1:91,1] = PR[GP1:90,1] + -0.264;
   1:  PR[GP1:91,2] = PR[GP1:90,2] + -35.509;
   1:L PR[91] 10mm/sec CNT100;
   1:  PR[GP1:91,1] = PR[GP1:90,1] + 1.314;
   1:  PR[GP1:91,2] = PR[GP1:90,2] + -36.651;
   1:  PR[GP1:91,3] = PR[GP1:90,3] + 81.435;
   1:L PR[91] 10mm/sec CNT100;
   1:  PR[GP1:91,1] = PR[GP1:90,1] + 1.861;
   1:  PR[GP1:91,2] = PR[GP1:90,2] + -36.808;
   1:L PR[91] 10mm/sec CNT100;
   1:  PR[GP1:91,1] = PR[GP1:90,1] + 14.266;
   1:  PR[GP1:91,2] = PR[GP1:90,2] + -39.646;
   1:L PR[91] 10mm/sec CNT100;
   1:  PR[GP1:91,1] = PR[GP1:90,1] + 15.154;
   1:  PR[GP1:91,2] = PR[GP1:90,2] + -39.705;
   1:L PR[91] 10mm/sec CNT100;
   1:  PR[GP1:91,1] = PR[GP1:90,1] + 16.207;
   1:  PR[GP1:91,2] = PR[GP1:90,2] + -39.560;
   1:L PR[91] 10mm/sec CNT100;
   1:  PR[GP1:91,1] = PR[GP1:90,1] + 28.367;
   1:  PR[GP1:91,2] = PR[GP1:90,2] + -38.378;
   1:L PR[91] 10mm/sec CNT100;
   1:  PR[GP1:91,1] = PR[GP1:90,1] + 29.664;
   1:  PR[GP1:91,2] = PR[GP1:90,2] + -37.905;
   1:L PR[91] 10mm/sec CNT100;
   1:  PR[GP1:91,1] = PR[GP1:90,1] + 40.074;
   1:  PR[GP1:91,2] = PR[GP1:90,2] + -33.327;
   1:L PR[91] 10mm/sec CNT100;
   1:  PR[GP1:91,1] = PR[GP1:90,1] + 41.481;
   1:  PR[GP1:91,2] = PR[GP1:90,2] + -32.444;
   1:L PR[91] 10mm/sec CNT100;
   1:  PR[GP1:91,1] = PR[GP1:90,1] + 42.793;
   1:  PR[GP1:91,2] = PR[GP1:90,2] + -31.166;
   1:L PR[91] 10mm/sec CNT100;
   1:  PR[GP1:91,1] = PR[GP1:90,1] + 50.693;
   1:  PR[GP1:91,2] = PR[GP1:90,2] + -23.980;
   1:L PR[91] 10mm/sec CNT100;
   1:  PR[GP1:91,1] = PR[GP1:90,1] + 51.812;
   1:  PR[GP1:91,2] = PR[GP1:90,2] + -22.245;
   1:L PR[91] 10mm/sec CNT100;
   1:  PR[GP1:91,1] = PR[GP1:90,1] + 56.662;
   1:  PR[GP1:91,2] = PR[GP1:90,2] + -13.477;
   1:L PR[91] 10mm/sec CNT100;
   1:  PR[GP1:91,1] = PR[GP1:90,1] + 57.395;
   1:  PR[GP1:91,2] = PR[GP1:90,2] + -11.486;
   1:L PR[91] 10mm/sec CNT100;
   1:  PR[GP1:91,1] = PR[GP1:90,1] + 57.646;
   1:  PR[GP1:91,2] = PR[GP1:90,2] + -9.275;
   1:L PR[91] 10mm/sec CNT100;
   1:  PR[GP1:91,1] = PR[GP1:90,1] + 59.278;
   1:  PR[GP1:91,2] = PR[GP1:90,2] + 0.296;
   1:L PR[91] 10mm/sec CNT100;
   1:  PR[GP1:91,1] = PR[GP1:90,1] + 59.031;
   1:  PR[GP1:91,2] = PR[GP1:90,2] + 2.485;
   1:L PR[91] 10mm/sec CNT100;
   1:  PR[GP1:91,1] = PR[GP1:90,1] + 57.393;
   1:  PR[GP1:91,2] = PR[GP1:90,2] + 12.047;
   1:L PR[91] 10mm/sec CNT100;
   1:  PR[GP1:91,1] = PR[GP1:90,1] + 56.655;
   1:  PR[GP1:91,2] = PR[GP1:90,2] + 14.055;
   1:L PR[91] 10mm/sec CNT100;
   1:  PR[GP1:91,1] = PR[GP1:90,1] + 51.784;
   1:  PR[GP1:91,2] = PR[GP1:90,2] + 22.838;
   1:L PR[91] 10mm/sec CNT100;
   1:  PR[GP1:91,1] = PR[GP1:90,1] + 50.659;
   1:  PR[GP1:91,2] = PR[GP1:90,2] + 24.583;
   1:L PR[91] 10mm/sec CNT100;
   1:  PR[GP1:91,1] = PR[GP1:90,1] + 49.305;
   1:  PR[GP1:91,2] = PR[GP1:90,2] + 25.908;
   1:L PR[91] 10mm/sec CNT100;
   1:  PR[GP1:91,1] = PR[GP1:90,1] + 41.431;
   1:  PR[GP1:91,2] = PR[GP1:90,2] + 33.035;
   1:L PR[91] 10mm/sec CNT100;
   1:  PR[GP1:91,1] = PR[GP1:90,1] + 40.016;
   1:  PR[GP1:91,2] = PR[GP1:90,2] + 33.923;
   1:L PR[91] 10mm/sec CNT100;
   1:  PR[GP1:91,1] = PR[GP1:90,1] + 29.565;
   1:  PR[GP1:91,2] = PR[GP1:90,2] + 38.489;
   1:L PR[91] 10mm/sec CNT100;
   1:  PR[GP1:91,1] = PR[GP1:90,1] + 28.256;
   1:  PR[GP1:91,2] = PR[GP1:90,2] + 38.967;
   1:L PR[91] 10mm/sec CNT100;
   1:  PR[GP1:91,1] = PR[GP1:90,1] + 27.021;
   1:  PR[GP1:91,2] = PR[GP1:90,2] + 39.142;
   1:L PR[91] 10mm/sec CNT100;
   1:  PR[GP1:91,1] = PR[GP1:90,1] + 15.032;
   1:  PR[GP1:91,2] = PR[GP1:90,2] + 40.256;
   1:L PR[91] 10mm/sec CNT100;
   1:  PR[GP1:91,1] = PR[GP1:90,1] + 14.136;
   1:  PR[GP1:91,2] = PR[GP1:90,2] + 40.196;
   1:L PR[91] 10mm/sec CNT100;
   1:  PR[GP1:91,1] = PR[GP1:90,1] + 1.528;
   1:  PR[GP1:91,2] = PR[GP1:90,2] + 37.218;
   1:L PR[91] 10mm/sec CNT100;
   1:  PR[GP1:91,1] = PR[GP1:90,1] + 1.073;
   1:  PR[GP1:91,2] = PR[GP1:90,2] + 37.088;
   1:L PR[91] 10mm/sec CNT100;
   1:  PR[GP1:91,1] = PR[GP1:90,1] + -0.263;
   1:  PR[GP1:91,2] = PR[GP1:90,2] + 36.387;
   1:L PR[91] 10mm/sec CNT100;
   1:  PR[GP1:91,1] = PR[GP1:90,1] + -1.596;
   1:  PR[GP1:91,2] = PR[GP1:90,2] + 37.088;
   1:L PR[91] 10mm/sec CNT100;
   1:  PR[GP1:91,1] = PR[GP1:90,1] + -2.049;
   1:  PR[GP1:91,2] = PR[GP1:90,2] + 37.218;
   1:L PR[91] 10mm/sec CNT100;
   1:  PR[GP1:91,1] = PR[GP1:90,1] + -14.661;
   1:  PR[GP1:91,2] = PR[GP1:90,2] + 40.196;
   1:L PR[91] 10mm/sec CNT100;
   1:  PR[GP1:91,1] = PR[GP1:90,1] + -15.547;
   1:  PR[GP1:91,2] = PR[GP1:90,2] + 40.254;
   1:L PR[91] 10mm/sec CNT100;
   1:  PR[GP1:91,1] = PR[GP1:90,1] + -16.602;
   1:  PR[GP1:91,2] = PR[GP1:90,2] + 40.108;
   1:L PR[91] 10mm/sec CNT100;
   1:  PR[GP1:91,1] = PR[GP1:90,1] + -28.803;
   1:  PR[GP1:91,2] = PR[GP1:90,2] + 38.961;
   1:L PR[91] 10mm/sec CNT100;
   1:  PR[GP1:91,1] = PR[GP1:90,1] + -30.096;
   1:  PR[GP1:91,2] = PR[GP1:90,2] + 38.488;
   1:L PR[91] 10mm/sec CNT100;
   1:  PR[GP1:91,1] = PR[GP1:90,1] + -40.547;
   1:  PR[GP1:91,2] = PR[GP1:90,2] + 33.918;
   1:L PR[91] 10mm/sec CNT100;
   1:  PR[GP1:91,1] = PR[GP1:90,1] + -41.962;
   1:  PR[GP1:91,2] = PR[GP1:90,2] + 33.026;
   1:L PR[91] 10mm/sec CNT100;
   1:  PR[GP1:91,1] = PR[GP1:90,1] + -43.276;
   1:  PR[GP1:91,2] = PR[GP1:90,2] + 31.743;
   1:L PR[91] 10mm/sec CNT100;
   1:  PR[GP1:91,1] = PR[GP1:90,1] + -51.209;
   1:  PR[GP1:91,2] = PR[GP1:90,2] + 24.560;
   1:L PR[91] 10mm/sec CNT100;
   1:  PR[GP1:91,1] = PR[GP1:90,1] + -52.316;
   1:  PR[GP1:91,2] = PR[GP1:90,2] + 22.834;
   1:L PR[91] 10mm/sec CNT100;
   1:  PR[GP1:91,1] = PR[GP1:90,1] + -57.187;
   1:  PR[GP1:91,2] = PR[GP1:90,2] + 14.035;
   1:L PR[91] 10mm/sec CNT100;
   1:  PR[GP1:91,1] = PR[GP1:90,1] + -57.923;
   1:  PR[GP1:91,2] = PR[GP1:90,2] + 12.007;
   1:L PR[91] 10mm/sec CNT100;
   1:  PR[GP1:91,1] = PR[GP1:90,1] + -58.165;
   1:  PR[GP1:91,2] = PR[GP1:90,2] + 9.844;
   1:L PR[91] 10mm/sec CNT100;
   1:  PR[GP1:91,1] = PR[GP1:90,1] + -59.805;
   1:  PR[GP1:91,2] = PR[GP1:90,2] + 0.261;
   1:L PR[91] 10mm/sec CNT100;
   1:  PR[GP1:91,1] = PR[GP1:90,1] + -59.566;
   1:  PR[GP1:91,2] = PR[GP1:90,2] + -1.880;
   1:L PR[91] 10mm/sec CNT100;
   1:  PR[GP1:91,1] = PR[GP1:90,1] + -57.936;
   1:  PR[GP1:91,2] = PR[GP1:90,2] + -11.413;
   1:L PR[91] 10mm/sec CNT100;
   1:  PR[GP1:91,1] = PR[GP1:90,1] + -57.194;
   1:  PR[GP1:91,2] = PR[GP1:90,2] + -13.457;
   1:L PR[91] 10mm/sec CNT100;
   1:  PR[GP1:91,1] = PR[GP1:90,1] + -52.343;
   1:  PR[GP1:91,2] = PR[GP1:90,2] + -22.240;
   1:L PR[91] 10mm/sec CNT100;
   1:  PR[GP1:91,1] = PR[GP1:90,1] + -51.230;
   1:  PR[GP1:91,2] = PR[GP1:90,2] + -23.978;
   1:L PR[91] 10mm/sec CNT100;
   1:  PR[GP1:91,1] = PR[GP1:90,1] + -49.874;
   1:  PR[GP1:91,2] = PR[GP1:90,2] + -25.308;
   1:L PR[91] 10mm/sec CNT100;
   1:  PR[GP1:91,1] = PR[GP1:90,1] + -42.032;
   1:  PR[GP1:91,2] = PR[GP1:90,2] + -32.423;
   1:L PR[91] 10mm/sec CNT100;
   1:  PR[GP1:91,1] = PR[GP1:90,1] + -40.606;
   1:  PR[GP1:91,2] = PR[GP1:90,2] + -33.322;
   1:L PR[91] 10mm/sec CNT100;
   1:  PR[GP1:91,1] = PR[GP1:90,1] + -30.195;
   1:  PR[GP1:91,2] = PR[GP1:90,2] + -37.903;
   1:L PR[91] 10mm/sec CNT100;
   1:  PR[GP1:91,1] = PR[GP1:90,1] + -28.888;
   1:  PR[GP1:91,2] = PR[GP1:90,2] + -38.382;
   1:L PR[91] 10mm/sec CNT100;
   1:  PR[GP1:91,1] = PR[GP1:90,1] + -27.646;
   1:  PR[GP1:91,2] = PR[GP1:90,2] + -38.559;
   1:L PR[91] 10mm/sec CNT100;
   1:  PR[GP1:91,1] = PR[GP1:90,1] + -15.696;
   1:  PR[GP1:91,2] = PR[GP1:90,2] + -39.706;
   1:L PR[91] 10mm/sec CNT100;
   1:  PR[GP1:91,1] = PR[GP1:90,1] + -14.792;
   1:  PR[GP1:91,2] = PR[GP1:90,2] + -39.646;
   1:L PR[91] 10mm/sec CNT100;
   1:  PR[GP1:91,1] = PR[GP1:90,1] + -2.387;
   1:  PR[GP1:91,2] = PR[GP1:90,2] + -36.808;
   1:L PR[91] 10mm/sec CNT100;
   1:  PR[GP1:91,1] = PR[GP1:90,1] + -1.841;
   1:  PR[GP1:91,2] = PR[GP1:90,2] + -36.651;
   1:L PR[91] 10mm/sec CNT100;
   1:  PR[GP1:91,1] = PR[GP1:90,1] + -0.264;
   1:  PR[GP1:91,2] = PR[GP1:90,2] + -35.727;
   1:L PR[91] 10mm/sec CNT100;
   1:  PR[GP1:91,1] = PR[GP1:90,1] + 1.059;
   1:  PR[GP1:91,2] = PR[GP1:90,2] + -36.720;
   1:  PR[GP1:91,3] = PR[GP1:90,3] + 82.045;
   1:L PR[91] 10mm/sec CNT100;
   1:  PR[GP1:91,1] = PR[GP1:90,1] + 1.486;
   1:  PR[GP1:91,2] = PR[GP1:90,2] + -36.843;
   1:L PR[91] 10mm/sec CNT100;
   1:  PR[GP1:91,1] = PR[GP1:90,1] + 14.090;
   1:  PR[GP1:91,2] = PR[GP1:90,2] + -39.727;
   1:L PR[91] 10mm/sec CNT100;
   1:  PR[GP1:91,1] = PR[GP1:90,1] + 14.854;
   1:  PR[GP1:91,2] = PR[GP1:90,2] + -39.777;
   1:L PR[91] 10mm/sec CNT100;
   1:  PR[GP1:91,1] = PR[GP1:90,1] + 15.771;
   1:  PR[GP1:91,2] = PR[GP1:90,2] + -39.651;
   1:L PR[91] 10mm/sec CNT100;
   1:  PR[GP1:91,1] = PR[GP1:90,1] + 28.150;
   1:  PR[GP1:91,2] = PR[GP1:90,2] + -38.448;
   1:L PR[91] 10mm/sec CNT100;
   1:  PR[GP1:91,1] = PR[GP1:90,1] + 29.320;
   1:  PR[GP1:91,2] = PR[GP1:90,2] + -38.021;
   1:L PR[91] 10mm/sec CNT100;
   1:  PR[GP1:91,1] = PR[GP1:90,1] + 39.929;
   1:  PR[GP1:91,2] = PR[GP1:90,2] + -33.355;
   1:L PR[91] 10mm/sec CNT100;
   1:  PR[GP1:91,1] = PR[GP1:90,1] + 41.226;
   1:  PR[GP1:91,2] = PR[GP1:90,2] + -32.542;
   1:L PR[91] 10mm/sec CNT100;
   1:  PR[GP1:91,1] = PR[GP1:90,1] + 42.438;
   1:  PR[GP1:91,2] = PR[GP1:90,2] + -31.360;
   1:L PR[91] 10mm/sec CNT100;
   1:  PR[GP1:91,1] = PR[GP1:90,1] + 50.506;
   1:  PR[GP1:91,2] = PR[GP1:90,2] + -24.022;
   1:L PR[91] 10mm/sec CNT100;
   1:  PR[GP1:91,1] = PR[GP1:90,1] + 51.550;
   1:  PR[GP1:91,2] = PR[GP1:90,2] + -22.402;
   1:L PR[91] 10mm/sec CNT100;
   1:  PR[GP1:91,1] = PR[GP1:90,1] + 56.508;
   1:  PR[GP1:91,2] = PR[GP1:90,2] + -13.441;
   1:L PR[91] 10mm/sec CNT100;
   1:  PR[GP1:91,1] = PR[GP1:90,1] + 57.195;
   1:  PR[GP1:91,2] = PR[GP1:90,2] + -11.572;
   1:L PR[91] 10mm/sec CNT100;
   1:  PR[GP1:91,1] = PR[GP1:90,1] + 57.431;
   1:  PR[GP1:91,2] = PR[GP1:90,2] + -9.495;
   1:L PR[91] 10mm/sec CNT100;
   1:  PR[GP1:91,1] = PR[GP1:90,1] + 59.101;
   1:  PR[GP1:91,2] = PR[GP1:90,2] + 0.296;
   1:L PR[91] 10mm/sec CNT100;
   1:  PR[GP1:91,1] = PR[GP1:90,1] + 58.868;
   1:  PR[GP1:91,2] = PR[GP1:90,2] + 2.354;
   1:L PR[91] 10mm/sec CNT100;
   1:  PR[GP1:91,1] = PR[GP1:90,1] + 57.194;
   1:  PR[GP1:91,2] = PR[GP1:90,2] + 12.135;
   1:L PR[91] 10mm/sec CNT100;
   1:  PR[GP1:91,1] = PR[GP1:90,1] + 56.501;
   1:  PR[GP1:91,2] = PR[GP1:90,2] + 14.019;
   1:L PR[91] 10mm/sec CNT100;
   1:  PR[GP1:91,1] = PR[GP1:90,1] + 51.522;
   1:  PR[GP1:91,2] = PR[GP1:90,2] + 22.996;
   1:L PR[91] 10mm/sec CNT100;
   1:  PR[GP1:91,1] = PR[GP1:90,1] + 50.471;
   1:  PR[GP1:91,2] = PR[GP1:90,2] + 24.625;
   1:L PR[91] 10mm/sec CNT100;
   1:  PR[GP1:91,1] = PR[GP1:90,1] + 49.208;
   1:  PR[GP1:91,2] = PR[GP1:90,2] + 25.863;
   1:L PR[91] 10mm/sec CNT100;
   1:  PR[GP1:91,1] = PR[GP1:90,1] + 41.174;
   1:  PR[GP1:91,2] = PR[GP1:90,2] + 33.133;
   1:L PR[91] 10mm/sec CNT100;
   1:  PR[GP1:91,1] = PR[GP1:90,1] + 39.869;
   1:  PR[GP1:91,2] = PR[GP1:90,2] + 33.952;
   1:L PR[91] 10mm/sec CNT100;
   1:  PR[GP1:91,1] = PR[GP1:90,1] + 29.219;
   1:  PR[GP1:91,2] = PR[GP1:90,2] + 38.605;
   1:L PR[91] 10mm/sec CNT100;
   1:  PR[GP1:91,1] = PR[GP1:90,1] + 28.037;
   1:  PR[GP1:91,2] = PR[GP1:90,2] + 39.037;
   1:L PR[91] 10mm/sec CNT100;
   1:  PR[GP1:91,1] = PR[GP1:90,1] + 26.922;
   1:  PR[GP1:91,2] = PR[GP1:90,2] + 39.195;
   1:L PR[91] 10mm/sec CNT100;
   1:  PR[GP1:91,1] = PR[GP1:90,1] + 14.730;
   1:  PR[GP1:91,2] = PR[GP1:90,2] + 40.328;
   1:L PR[91] 10mm/sec CNT100;
   1:  PR[GP1:91,1] = PR[GP1:90,1] + 13.957;
   1:  PR[GP1:91,2] = PR[GP1:90,2] + 40.276;
   1:L PR[91] 10mm/sec CNT100;
   1:  PR[GP1:91,1] = PR[GP1:90,1] + 1.147;
   1:  PR[GP1:91,2] = PR[GP1:90,2] + 37.251;
   1:L PR[91] 10mm/sec CNT100;
   1:  PR[GP1:91,1] = PR[GP1:90,1] + 0.815;
   1:  PR[GP1:91,2] = PR[GP1:90,2] + 37.155;
   1:L PR[91] 10mm/sec CNT100;
   1:  PR[GP1:91,1] = PR[GP1:90,1] + -0.262;
   1:  PR[GP1:91,2] = PR[GP1:90,2] + 36.590;
   1:L PR[91] 10mm/sec CNT100;
   1:  PR[GP1:91,1] = PR[GP1:90,1] + -1.337;
   1:  PR[GP1:91,2] = PR[GP1:90,2] + 37.156;
   1:L PR[91] 10mm/sec CNT100;
   1:  PR[GP1:91,1] = PR[GP1:90,1] + -1.668;
   1:  PR[GP1:91,2] = PR[GP1:90,2] + 37.251;
   1:L PR[91] 10mm/sec CNT100;
   1:  PR[GP1:91,1] = PR[GP1:90,1] + -14.482;
   1:  PR[GP1:91,2] = PR[GP1:90,2] + 40.276;
   1:L PR[91] 10mm/sec CNT100;
   1:  PR[GP1:91,1] = PR[GP1:90,1] + -15.245;
   1:  PR[GP1:91,2] = PR[GP1:90,2] + 40.326;
   1:L PR[91] 10mm/sec CNT100;
   1:  PR[GP1:91,1] = PR[GP1:90,1] + -16.163;
   1:  PR[GP1:91,2] = PR[GP1:90,2] + 40.199;
   1:L PR[91] 10mm/sec CNT100;
